LIN {X 0,Y 262.907,Z 862.683,A -85,B 0,C 180,E1 12997.239,E2 12997.239} C_VEL
LIN {X 0,Y 257.148,Z 985.55,A -85,B 0,C 180,E1 12992.155,E2 12992.155} C_VEL
LIN {X 0,Y 256.421,Z 1011.983,A -85,B 0,C 180,E1 12990.929,E2 12990.929} C_VEL
LIN {X 0,Y 255.607,Z 1029.219,A -85,B 0,C 180,E1 12989.732,E2 12989.732} C_VEL
LIN {X 0,Y 254.567,Z 1046.159,A -85,B 0,C 180,E1 12988.115,E2 12988.115} C_VEL
LIN {X 0,Y 253.439,Z 1061.43,A -85,B 0,C 180,E1 12986.217,E2 12986.217} C_VEL
LIN {X 0,Y 252.31,Z 1075.854,A -85,B 0,C 180,E1 12983.96,E2 12983.96} C_VEL
LIN {X 0,Y 251.242,Z 1089.802,A -85,B 0,C 180,E1 12981.227,E2 12981.227} C_VEL
LIN {X 0,Y 250.502,Z 1101.467,A -85,B 0,C 180,E1 12978.375,E2 12978.375} C_VEL
LIN {X 0,Y 250.09,Z 1111.696,A -85,B 0,C 180,E1 12975.295,E2 12975.295} C_VEL
LIN {X 0,Y 250.084,Z 1120.327,A -85,B 0,C 180,E1 12971.994,E2 12971.994} C_VEL
LIN {X 0,Y 250.563,Z 1126.995,A -85,B 0,C 180,E1 12968.717,E2 12968.717} C_VEL
LIN {X 0,Y 251.586,Z 1131.816,A -85,B 0,C 180,E1 12965.468,E2 12965.468} C_VEL
LIN {X 0,Y 253.23,Z 1135.281,A -85,B 0,C 180,E1 12962.258,E2 12962.258} C_VEL
LIN {X 0,Y 255.925,Z 1137.41,A -85,B 0,C 180,E1 12958.652,E2 12958.652} C_VEL
LIN {X 0,Y 259.509,Z 1137.615,A -85,B 0,C 180,E1 12955.133,E2 12955.133} C_VEL
LIN {X 0,Y 263.997,Z 1136.033,A -85,B 0,C 180,E1 12951.72,E2 12951.72} C_VEL
LIN {X 0,Y 265.449,Z 1135.191,A -85,B 0,C 180,E1 12950.758,E2 12950.758} C_VEL
LIN {X 0,Y 267.144,Z 1133.765,A -85,B 0,C 180,E1 12949.03,E2 12949.03} C_VEL
LIN {X 0,Y 268.599,Z 1130.246,A -85,B 0,C 180,E1 12945.292,E2 12945.292} C_VEL
LIN {X 0,Y 270.654,Z 1127.621,A -85,B 0,C 180,E1 12943.679,E2 12943.679} C_VEL
LIN {X 0,Y 271.079,Z 1127.193,A -85,B 0,C 180,E1 12943.483,E2 12943.483} C_VEL
LIN {X 0,Y 278.019,Z 1119.744,A -85,B 0,C 180,E1 12940.674,E2 12940.674} C_VEL
LIN {X 0,Y 285.046,Z 1110.662,A -85,B 0,C 180,E1 12938.167,E2 12938.167} C_VEL
LIN {X 0,Y 291.992,Z 1100.144,A -85,B 0,C 180,E1 12935.948,E2 12935.948} C_VEL
LIN {X 0,Y 298.978,Z 1087.604,A -85,B 0,C 180,E1 12933.906,E2 12933.906} C_VEL
LIN {X 0,Y 305.649,Z 1073.127,A -85,B 0,C 180,E1 12932.104,E2 12932.104} C_VEL
LIN {X 0,Y 310.7,Z 1059.737,A -85,B 0,C 180,E1 12930.816,E2 12930.816} C_VEL
LIN {X 0,Y 314.858,Z 1046.143,A -85,B 0,C 180,E1 12929.775,E2 12929.775} C_VEL
LIN {X 0,Y 318.495,Z 1031.06,A -85,B 0,C 180,E1 12928.863,E2 12928.863} C_VEL
LIN {X 0,Y 324.296,Z 999.248,A -85,B 0,C 180,E1 12927.506,E2 12927.506} C_VEL
LIN {X 0,Y 338.694,Z 926.288,A -85,B 0,C 180,E1 12925.071,E2 12925.071} C_VEL
LIN {X 0,Y 330.952,Z 955.979,A -85,B 0,C 180,E1 12923.859,E2 12923.859} C_VEL
LIN {X 0,Y 322.137,Z 991.386,A -85,B 0,C 180,E1 12922.542,E2 12922.542} C_VEL
LIN {X 0,Y 313.495,Z 1027.366,A -85,B 0,C 180,E1 12920.786,E2 12920.786} C_VEL
LIN {X 0,Y 308.225,Z 1048.269,A -85,B 0,C 180,E1 12919.544,E2 12919.544} C_VEL
LIN {X 0,Y 302.397,Z 1065.839,A -85,B 0,C 180,E1 12918.208,E2 12918.208} C_VEL
LIN {X 0,Y 295.952,Z 1082.262,A -85,B 0,C 180,E1 12916.721,E2 12916.721} C_VEL
LIN {X 0,Y 289.029,Z 1097.291,A -85,B 0,C 180,E1 12915.024,E2 12915.024} C_VEL
LIN {X 0,Y 281.432,Z 1112.235,A -85,B 0,C 180,E1 12912.868,E2 12912.868} C_VEL
LIN {X 0,Y 273.14,Z 1127.155,A -85,B 0,C 180,E1 12910.108,E2 12910.108} C_VEL
LIN {X 0,Y 265.471,Z 1140.112,A -85,B 0,C 180,E1 12907.054,E2 12907.054} C_VEL
LIN {X 0,Y 258.017,Z 1152.256,A -85,B 0,C 180,E1 12903.383,E2 12903.383} C_VEL
LIN {X 0,Y 251.919,Z 1162.119,A -85,B 0,C 180,E1 12899.479,E2 12899.479} C_VEL
LIN {X 0,Y 247.143,Z 1170.061,A -85,B 0,C 180,E1 12895.391,E2 12895.391} C_VEL
LIN {X 0,Y 243.863,Z 1176.091,A -85,B 0,C 180,E1 12891.147,E2 12891.147} C_VEL
LIN {X 0,Y 242.039,Z 1180.61,A -85,B 0,C 180,E1 12886.558,E2 12886.558} C_VEL
LIN {X 0,Y 241.078,Z 1189.876,A -85,B 0,C 180,E1 12881.965,E2 12881.965} C_VEL
LIN {X 0,Y 240.853,Z 1196.891,A -85,B 0,C 180,E1 12877.631,E2 12877.631} C_VEL
LIN {X 0,Y 240.925,Z 1201.889,A -85,B 0,C 180,E1 12873.566,E2 12873.566} C_VEL
LIN {X 0,Y 240.878,Z 1205.148,A -85,B 0,C 180,E1 12869.997,E2 12869.997} C_VEL
LIN {X 0,Y 240.501,Z 1207.636,A -85,B 0,C 180,E1 12865.944,E2 12865.944} C_VEL
LIN {X 0,Y 240.266,Z 1209.075,A -85,B 0,C 180,E1 12860.898,E2 12860.898} C_VEL
LIN {X 0,Y 241.096,Z 1209.016,A -85,B 0,C 180,E1 12855.588,E2 12855.588} C_VEL
LIN {X 0,Y 243.908,Z 1207.154,A -85,B 0,C 180,E1 12849.855,E2 12849.855} C_VEL
LIN {X 0,Y 249.522,Z 1203.368,A -85,B 0,C 180,E1 12843.842,E2 12843.842} C_VEL
LIN {X 0,Y 258.306,Z 1197.619,A -85,B 0,C 180,E1 12837.97,E2 12837.97} C_VEL
LIN {X 0,Y 270.003,Z 1190.061,A -85,B 0,C 180,E1 12832.6,E2 12832.6} C_VEL
LIN {X 0,Y 285.633,Z 1180.278,A -85,B 0,C 180,E1 12827.495,E2 12827.495} C_VEL
LIN {X 0,Y 303.551,Z 1169.347,A -85,B 0,C 180,E1 12823.252,E2 12823.252} C_VEL
LIN {X 0,Y 286.385,Z 1177.494,A -85,B 0,C 180,E1 12818.941,E2 12818.941} C_VEL
LIN {X 0,Y 272.266,Z 1183.771,A -85,B 0,C 180,E1 12814.191,E2 12814.191} C_VEL
LIN {X 0,Y 260.321,Z 1188.527,A -85,B 0,C 180,E1 12808.698,E2 12808.698} C_VEL
LIN {X 0,Y 251.821,Z 1191.239,A -85,B 0,C 180,E1 12803.152,E2 12803.152} C_VEL
LIN {X 0,Y 246.032,Z 1192.182,A -85,B 0,C 180,E1 12797.507,E2 12797.507} C_VEL
LIN {X 0,Y 242.552,Z 1191.319,A -85,B 0,C 180,E1 12791.9,E2 12791.9} C_VEL
LIN {X 0,Y 240.867,Z 1188.892,A -85,B 0,C 180,E1 12786.44,E2 12786.44} C_VEL
LIN {X 0,Y 240.315,Z 1185.407,A -85,B 0,C 180,E1 12781.674,E2 12781.674} C_VEL
LIN {X 0,Y 240.198,Z 1180.652,A -85,B 0,C 180,E1 12777.142,E2 12777.142} C_VEL
LIN {X 0,Y 240.391,Z 1174.513,A -85,B 0,C 180,E1 12772.597,E2 12772.597} C_VEL
LIN {X 0,Y 241.092,Z 1166.593,A -85,B 0,C 180,E1 12768.037,E2 12768.037} C_VEL
LIN {X 0,Y 242.519,Z 1156.908,A -85,B 0,C 180,E1 12763.478,E2 12763.478} C_VEL
LIN {X 0,Y 244.727,Z 1145.903,A -85,B 0,C 180,E1 12759.184,E2 12759.184} C_VEL
LIN {X 0,Y 247.867,Z 1132.744,A -85,B 0,C 180,E1 12754.946,E2 12754.946} C_VEL
LIN {X 0,Y 251.721,Z 1118.125,A -85,B 0,C 180,E1 12751.019,E2 12751.019} C_VEL
LIN {X 0,Y 256.476,Z 1101.03,A -85,B 0,C 180,E1 12747.193,E2 12747.193} C_VEL
LIN {X 0,Y 261.576,Z 1082.796,A -85,B 0,C 180,E1 12743.808,E2 12743.808} C_VEL
LIN {X 0,Y 266.72,Z 1063.992,A -85,B 0,C 180,E1 12740.9,E2 12740.9} C_VEL
LIN {X 0,Y 272.079,Z 1043.302,A -85,B 0,C 180,E1 12738.25,E2 12738.25} C_VEL
LIN {X 0,Y 277.383,Z 1021.009,A -85,B 0,C 180,E1 12735.923,E2 12735.923} C_VEL
LIN {X 0,Y 282.447,Z 997.128,A -85,B 0,C 180,E1 12733.919,E2 12733.919} C_VEL
LIN {X 0,Y 286.934,Z 972.487,A -85,B 0,C 180,E1 12732.294,E2 12732.294} C_VEL
LIN {X 0,Y 290.636,Z 947.66,A -85,B 0,C 180,E1 12731.044,E2 12731.044} C_VEL
LIN {X 0,Y 297.427,Z 889.487,A -85,B 0,C 180,E1 12728.954,E2 12728.954} C_VEL
LIN {X 0,Y 310.27,Z 781.665,A -85,B 0,C 180,E1 12725.402,E2 12725.402} C_VEL
LIN {X 0,Y 296.592,Z 756.31,A -85,B 0,C 180,E1 12722.045,E2 12722.045} C_VEL
LIN {X 0,Y 283.156,Z 732.602,A -85,B 0,C 180,E1 12718.388,E2 12718.388} C_VEL
LIN {X 0,Y 271.277,Z 712.791,A -85,B 0,C 180,E1 12714.82,E2 12714.82} C_VEL
LIN {X 0,Y 260.212,Z 695.463,A -85,B 0,C 180,E1 12711.177,E2 12711.177} C_VEL
LIN {X 0,Y 252.89,Z 684.704,A -85,B 0,C 180,E1 12708.562,E2 12708.562} C_VEL
LIN {X 0,Y 250.262,Z 680.677,A -85,B 0,C 180,E1 12707.56,E2 12707.56} C_VEL
LIN {X 0,Y 247.641,Z 676.731,A -85,B 0,C 180,E1 12706.541,E2 12706.541} C_VEL
LIN {X 0,Y 246.731,Z 675.484,A -85,B 0,C 180,E1 12706.19,E2 12706.19} C_VEL
LIN {X 0,Y 244.47,Z 672.459,A -85,B 0,C 180,E1 12705.299,E2 12705.299} C_VEL
LIN {X 0,Y 243.869,Z 670.279,A -85,B 0,C 180,E1 12704.912,E2 12704.912} C_VEL
LIN {X 0,Y 243.87,Z 670.278,A -85,B 0,C 180,E1 12699.919,E2 12699.919} C_VEL
LIN {X 0,Y 243.842,Z 670.293,A -85,B 0,C 180,E1 12694.943,E2 12694.943} C_VEL
LIN {X 0,Y 243.858,Z 670.294,A -85,B 0,C 180,E1 12689.533,E2 12689.533} C_VEL
LIN {X 0,Y 243.883,Z 670.266,A -85,B 0,C 180,E1 12684.592,E2 12684.592} C_VEL
LIN {X 0,Y 243.852,Z 670.26,A -85,B 0,C 180,E1 12679.732,E2 12679.732} C_VEL
LIN {X 0,Y 243.847,Z 670.293,A -85,B 0,C 180,E1 12674.473,E2 12674.473} C_VEL
LIN {X 0,Y 243.873,Z 670.284,A -85,B 0,C 180,E1 12669.357,E2 12669.357} C_VEL
LIN {X 0,Y 243.901,Z 670.438,A -85,B 0,C 180,E1 12664.735,E2 12664.735} C_VEL
LIN {X 0,Y 251.948,Z 691.844,A -85,B 0,C 180,E1 12660.525,E2 12660.525} C_VEL
LIN {X 0,Y 259.45,Z 713.889,A -85,B 0,C 180,E1 12656.561,E2 12656.561} C_VEL
LIN {X 0,Y 265.405,Z 734.117,A -85,B 0,C 180,E1 12653.205,E2 12653.205} C_VEL
LIN {X 0,Y 268.217,Z 745.033,A -85,B 0,C 180,E1 12651.501,E2 12651.501} C_VEL
LIN {X 0,Y 263.398,Z 787.814,A -85,B 0,C 180,E1 12646.466,E2 12646.466} C_VEL
LIN {X 0,Y 258.769,Z 832.439,A -85,B 0,C 180,E1 12641.187,E2 12641.187} C_VEL
LIN {X 0,Y 256.454,Z 854.436,A -85,B 0,C 180,E1 12638.589,E2 12638.589} C_VEL
LIN {X 0,Y 255.062,Z 863.549,A -85,B 0,C 180,E1 12637.603,E2 12637.603} C_VEL
LIN {X 0,Y 249.206,Z 985.599,A -85,B 0,C 180,E1 12632.372,E2 12632.372} C_VEL
LIN {X 0,Y 248.442,Z 1012.462,A -85,B 0,C 180,E1 12631.085,E2 12631.085} C_VEL
LIN {X 0,Y 247.567,Z 1030.453,A -85,B 0,C 180,E1 12629.781,E2 12629.781} C_VEL
LIN {X 0,Y 246.475,Z 1047.618,A -85,B 0,C 180,E1 12628.066,E2 12628.066} C_VEL
LIN {X 0,Y 245.276,Z 1063.53,A -85,B 0,C 180,E1 12625.985,E2 12625.985} C_VEL
LIN {X 0,Y 244.151,Z 1077.714,A -85,B 0,C 180,E1 12623.656,E2 12623.656} C_VEL
LIN {X 0,Y 243.108,Z 1091.585,A -85,B 0,C 180,E1 12620.823,E2 12620.823} C_VEL
LIN {X 0,Y 242.37,Z 1103.934,A -85,B 0,C 180,E1 12617.653,E2 12617.653} C_VEL
LIN {X 0,Y 242.052,Z 1113.48,A -85,B 0,C 180,E1 12614.589,E2 12614.589} C_VEL
LIN {X 0,Y 242.18,Z 1122.496,A -85,B 0,C 180,E1 12610.943,E2 12610.943} C_VEL
LIN {X 0,Y 242.922,Z 1129.293,A -85,B 0,C 180,E1 12607.295,E2 12607.295} C_VEL
LIN {X 0,Y 244.855,Z 1135.134,A -85,B 0,C 180,E1 12602.804,E2 12602.804} C_VEL
LIN {X 0,Y 247.469,Z 1138.004,A -85,B 0,C 180,E1 12599.069,E2 12599.069} C_VEL
LIN {X 0,Y 251.021,Z 1138.959,A -85,B 0,C 180,E1 12595.426,E2 12595.426} C_VEL
LIN {X 0,Y 255.522,Z 1138.14,A -85,B 0,C 180,E1 12591.897,E2 12591.897} C_VEL
LIN {X 0,Y 260.921,Z 1135.403,A -85,B 0,C 180,E1 12588.501,E2 12588.501} C_VEL
LIN {X 0,Y 267.191,Z 1130.78,A -85,B 0,C 180,E1 12585.253,E2 12585.253} C_VEL
LIN {X 0,Y 271.079,Z 1127.193,A -85,B 0,C 180,E1 12583.483,E2 12583.483} C_VEL
LIN {X 0,Y 273.484,Z 1124.348,A -85,B 0,C 180,E1 12582.046,E2 12582.046} C_VEL
LIN {X 0,Y 276.801,Z 1117.935,A -85,B 0,C 180,E1 12578.641,E2 12578.641} C_VEL
LIN {X 0,Y 279.108,Z 1114.254,A -85,B 0,C 180,E1 12577.323,E2 12577.323} C_VEL
LIN {X 0,Y 280.012,Z 1113.013,A -85,B 0,C 180,E1 12576.996,E2 12576.996} C_VEL
LIN {X 0,Y 287.643,Z 1102.313,A -85,B 0,C 180,E1 12574.683,E2 12574.683} C_VEL
LIN {X 0,Y 295.58,Z 1088.93,A -85,B 0,C 180,E1 12572.496,E2 12572.496} C_VEL
LIN {X 0,Y 302.679,Z 1074.368,A -85,B 0,C 180,E1 12570.698,E2 12570.698} C_VEL
LIN {X 0,Y 308.206,Z 1060.379,A -85,B 0,C 180,E1 12569.376,E2 12569.376} C_VEL
LIN {X 0,Y 312.574,Z 1046.756,A -85,B 0,C 180,E1 12568.354,E2 12568.354} C_VEL
LIN {X 0,Y 316.312,Z 1031.971,A -85,B 0,C 180,E1 12567.477,E2 12567.477} C_VEL
LIN {X 0,Y 322.674,Z 999.089,A -85,B 0,C 180,E1 12566.094,E2 12566.094} C_VEL
LIN {X 0,Y 329.477,Z 965.638,A -85,B 0,C 180,E1 12564.944,E2 12564.944} C_VEL
LIN {X 0,Y 320.95,Z 998.547,A -85,B 0,C 180,E1 12563.705,E2 12563.705} C_VEL
LIN {X 0,Y 310.763,Z 1038.509,A -85,B 0,C 180,E1 12561.704,E2 12561.704} C_VEL
LIN {X 0,Y 304.982,Z 1056.587,A -85,B 0,C 180,E1 12560.537,E2 12560.537} C_VEL
LIN {X 0,Y 297.577,Z 1075.428,A -85,B 0,C 180,E1 12558.963,E2 12558.963} C_VEL
LIN {X 0,Y 289.988,Z 1091.402,A -85,B 0,C 180,E1 12557.4,E2 12557.4} C_VEL
LIN {X 0,Y 281.3,Z 1107.424,A -85,B 0,C 180,E1 12555.304,E2 12555.304} C_VEL
LIN {X 0,Y 272.98,Z 1121.409,A -85,B 0,C 180,E1 12552.94,E2 12552.94} C_VEL
LIN {X 0,Y 264.299,Z 1134.834,A -85,B 0,C 180,E1 12550.022,E2 12550.022} C_VEL
LIN {X 0,Y 256.114,Z 1146.895,A -85,B 0,C 180,E1 12546.674,E2 12546.674} C_VEL
LIN {X 0,Y 248.363,Z 1157.914,A -85,B 0,C 180,E1 12542.643,E2 12542.643} C_VEL
LIN {X 0,Y 242.49,Z 1166.352,A -85,B 0,C 180,E1 12538.555,E2 12538.555} C_VEL
LIN {X 0,Y 237.831,Z 1173.199,A -85,B 0,C 180,E1 12534.063,E2 12534.063} C_VEL
LIN {X 0,Y 235.02,Z 1177.94,A -85,B 0,C 180,E1 12529.636,E2 12529.636} C_VEL
LIN {X 0,Y 233.992,Z 1180.433,A -85,B 0,C 180,E1 12526.25,E2 12526.25} C_VEL
LIN {X 0,Y 233.086,Z 1189.823,A -85,B 0,C 180,E1 12521.377,E2 12521.377} C_VEL
LIN {X 0,Y 232.929,Z 1196.73,A -85,B 0,C 180,E1 12516.9,E2 12516.9} C_VEL
LIN {X 0,Y 233.016,Z 1201.587,A -85,B 0,C 180,E1 12512.702,E2 12512.702} C_VEL
LIN {X 0,Y 232.885,Z 1204.73,A -85,B 0,C 180,E1 12509.013,E2 12509.013} C_VEL
LIN {X 0,Y 232.433,Z 1207.231,A -85,B 0,C 180,E1 12504.566,E2 12504.566} C_VEL
LIN {X 0,Y 232.386,Z 1208.487,A -85,B 0,C 180,E1 12499.335,E2 12499.335} C_VEL
LIN {X 0,Y 233.79,Z 1208.316,A -85,B 0,C 180,E1 12493.601,E2 12493.601} C_VEL
LIN {X 0,Y 237.606,Z 1206.216,A -85,B 0,C 180,E1 12487.481,E2 12487.481} C_VEL
LIN {X 0,Y 244.668,Z 1202.141,A -85,B 0,C 180,E1 12481.166,E2 12481.166} C_VEL
LIN {X 0,Y 254.823,Z 1196.35,A -85,B 0,C 180,E1 12475.319,E2 12475.319} C_VEL
LIN {X 0,Y 268.434,Z 1188.583,A -85,B 0,C 180,E1 12469.876,E2 12469.876} C_VEL
LIN {X 0,Y 285.564,Z 1178.951,A -85,B 0,C 180,E1 12464.982,E2 12464.982} C_VEL
LIN {X 0,Y 293.426,Z 1174.599,A -85,B 0,C 180,E1 12463.175,E2 12463.175} C_VEL
LIN {X 0,Y 276.489,Z 1181.641,A -85,B 0,C 180,E1 12458.733,E2 12458.733} C_VEL
LIN {X 0,Y 262.024,Z 1187.123,A -85,B 0,C 180,E1 12453.6,E2 12453.6} C_VEL
LIN {X 0,Y 250.761,Z 1190.751,A -85,B 0,C 180,E1 12448.073,E2 12448.073} C_VEL
LIN {X 0,Y 242.54,Z 1192.595,A -85,B 0,C 180,E1 12442.294,E2 12442.294} C_VEL
LIN {X 0,Y 237.092,Z 1192.604,A -85,B 0,C 180,E1 12436.418,E2 12436.418} C_VEL
LIN {X 0,Y 233.992,Z 1190.949,A -85,B 0,C 180,E1 12430.593,E2 12430.593} C_VEL
LIN {X 0,Y 232.645,Z 1187.943,A -85,B 0,C 180,E1 12425.184,E2 12425.184} C_VEL
LIN {X 0,Y 232.26,Z 1183.944,A -85,B 0,C 180,E1 12420.499,E2 12420.499} C_VEL
LIN {X 0,Y 232.221,Z 1178.664,A -85,B 0,C 180,E1 12415.808,E2 12415.808} C_VEL
LIN {X 0,Y 232.535,Z 1172.134,A -85,B 0,C 180,E1 12411.35,E2 12411.35} C_VEL
LIN {X 0,Y 233.498,Z 1163.129,A -85,B 0,C 180,E1 12406.383,E2 12406.383} C_VEL
LIN {X 0,Y 235.289,Z 1152.65,A -85,B 0,C 180,E1 12401.677,E2 12401.677} C_VEL
LIN {X 0,Y 237.924,Z 1140.682,A -85,B 0,C 180,E1 12397.261,E2 12397.261} C_VEL
LIN {X 0,Y 241.318,Z 1127.356,A -85,B 0,C 180,E1 12393.158,E2 12393.158} C_VEL
LIN {X 0,Y 245.76,Z 1111.304,A -85,B 0,C 180,E1 12389.031,E2 12389.031} C_VEL
LIN {X 0,Y 250.677,Z 1094.143,A -85,B 0,C 180,E1 12385.366,E2 12385.366} C_VEL
LIN {X 0,Y 255.878,Z 1075.916,A -85,B 0,C 180,E1 12382.129,E2 12382.129} C_VEL
LIN {X 0,Y 261.644,Z 1054.884,A -85,B 0,C 180,E1 12379.058,E2 12379.058} C_VEL
LIN {X 0,Y 267.378,Z 1032.375,A -85,B 0,C 180,E1 12376.381,E2 12376.381} C_VEL
LIN {X 0,Y 272.795,Z 1009.003,A -85,B 0,C 180,E1 12374.143,E2 12374.143} C_VEL
LIN {X 0,Y 277.725,Z 984.619,A -85,B 0,C 180,E1 12372.289,E2 12372.289} C_VEL
LIN {X 0,Y 281.98,Z 959.598,A -85,B 0,C 180,E1 12370.819,E2 12370.819} C_VEL
LIN {X 0,Y 285.461,Z 933.761,A -85,B 0,C 180,E1 12369.699,E2 12369.699} C_VEL
LIN {X 0,Y 303.575,Z 784.388,A -85,B 0,C 180,E1 12364.573,E2 12364.573} C_VEL
LIN {X 0,Y 288.726,Z 756.795,A -85,B 0,C 180,E1 12360.778,E2 12360.778} C_VEL
LIN {X 0,Y 274.471,Z 731.706,A -85,B 0,C 180,E1 12356.682,E2 12356.682} C_VEL
LIN {X 0,Y 262.767,Z 712.512,A -85,B 0,C 180,E1 12352.971,E2 12352.971} C_VEL
LIN {X 0,Y 252.332,Z 696.388,A -85,B 0,C 180,E1 12349.325,E2 12349.325} C_VEL
LIN {X 0,Y 245.659,Z 686.526,A -85,B 0,C 180,E1 12346.8,E2 12346.8} C_VEL
LIN {X 0,Y 242.421,Z 681.711,A -85,B 0,C 180,E1 12345.493,E2 12345.493} C_VEL
LIN {X 0,Y 239.862,Z 677.766,A -85,B 0,C 180,E1 12344.395,E2 12344.395} C_VEL
LIN {X 0,Y 239.036,Z 676.628,A -85,B 0,C 180,E1 12344.044,E2 12344.044} C_VEL
LIN {X 0,Y 236.628,Z 673.64,A -85,B 0,C 180,E1 12343.038,E2 12343.038} C_VEL
LIN {X 0,Y 235.942,Z 671.261,A -85,B 0,C 180,E1 12342.593,E2 12342.593} C_VEL
LIN {X 0,Y 235.928,Z 671.262,A -85,B 0,C 180,E1 12337.308,E2 12337.308} C_VEL
LIN {X 0,Y 235.879,Z 671.259,A -85,B 0,C 180,E1 12332.19,E2 12332.19} C_VEL
LIN {X 0,Y 235.934,Z 671.254,A -85,B 0,C 180,E1 12327.331,E2 12327.331} C_VEL
LIN {X 0,Y 235.949,Z 671.278,A -85,B 0,C 180,E1 12322.21,E2 12322.21} C_VEL
LIN {X 0,Y 235.905,Z 671.261,A -85,B 0,C 180,E1 12316.772,E2 12316.772} C_VEL
LIN {X 0,Y 235.916,Z 671.281,A -85,B 0,C 180,E1 12311.469,E2 12311.469} C_VEL
LIN {X 0,Y 235.952,Z 671.272,A -85,B 0,C 180,E1 12306.53,E2 12306.53} C_VEL
LIN {X 0,Y 235.972,Z 671.45,A -85,B 0,C 180,E1 12305.849,E2 12305.849} C_VEL
LIN {X 0,Y 243.869,Z 692.127,A -85,B 0,C 180,E1 12301.605,E2 12301.605} C_VEL
LIN {X 0,Y 251.152,Z 713.391,A -85,B 0,C 180,E1 12297.628,E2 12297.628} C_VEL
LIN {X 0,Y 257.574,Z 734.773,A -85,B 0,C 180,E1 12293.981,E2 12293.981} C_VEL
LIN {X 0,Y 260.697,Z 747.225,A -85,B 0,C 180,E1 12291.996,E2 12291.996} C_VEL
LIN {X 0,Y 255.647,Z 790.521,A -85,B 0,C 180,E1 12286.812,E2 12286.812} C_VEL
LIN {X 0,Y 250.873,Z 835.148,A -85,B 0,C 180,E1 12281.416,E2 12281.416} C_VEL
LIN {X 0,Y 248.798,Z 854.259,A -85,B 0,C 180,E1 12279.114,E2 12279.114} C_VEL
LIN {X 0,Y 247.229,Z 864.336,A -85,B 0,C 180,E1 12277.99,E2 12277.99} C_VEL
LIN {X 0,Y 241.255,Z 985.467,A -85,B 0,C 180,E1 12272.577,E2 12272.577} C_VEL
LIN {X 0,Y 240.415,Z 1013.694,A -85,B 0,C 180,E1 12271.16,E2 12271.16} C_VEL
LIN {X 0,Y 239.54,Z 1031.22,A -85,B 0,C 180,E1 12269.846,E2 12269.846} C_VEL
LIN {X 0,Y 238.384,Z 1048.948,A -85,B 0,C 180,E1 12268.013,E2 12268.013} C_VEL
LIN {X 0,Y 237.109,Z 1065.635,A -85,B 0,C 180,E1 12265.738,E2 12265.738} C_VEL
LIN {X 0,Y 235.94,Z 1080.241,A -85,B 0,C 180,E1 12263.205,E2 12263.205} C_VEL
LIN {X 0,Y 235.048,Z 1092.259,A -85,B 0,C 180,E1 12260.642,E2 12260.642} C_VEL
LIN {X 0,Y 234.333,Z 1104.572,A -85,B 0,C 180,E1 12257.373,E2 12257.373} C_VEL
LIN {X 0,Y 234.04,Z 1114.526,A -85,B 0,C 180,E1 12254.089,E2 12254.089} C_VEL
LIN {X 0,Y 234.256,Z 1123.525,A -85,B 0,C 180,E1 12250.322,E2 12250.322} C_VEL
LIN {X 0,Y 235.12,Z 1130.307,A -85,B 0,C 180,E1 12246.588,E2 12246.588} C_VEL
LIN {X 0,Y 237.163,Z 1135.991,A -85,B 0,C 180,E1 12242.169,E2 12242.169} C_VEL
LIN {X 0,Y 240.07,Z 1139.072,A -85,B 0,C 180,E1 12238.23,E2 12238.23} C_VEL
LIN {X 0,Y 243.806,Z 1140.18,A -85,B 0,C 180,E1 12234.582,E2 12234.582} C_VEL
LIN {X 0,Y 248.941,Z 1139.436,A -85,B 0,C 180,E1 12230.75,E2 12230.75} C_VEL
LIN {X 0,Y 254.74,Z 1136.817,A -85,B 0,C 180,E1 12227.298,E2 12227.298} C_VEL
LIN {X 0,Y 261.427,Z 1132.299,A -85,B 0,C 180,E1 12224.011,E2 12224.011} C_VEL
LIN {X 0,Y 268.53,Z 1126.01,A -85,B 0,C 180,E1 12221.035,E2 12221.035} C_VEL
LIN {X 0,Y 276.036,Z 1117.959,A -85,B 0,C 180,E1 12218.312,E2 12218.312} C_VEL
LIN {X 0,Y 280.012,Z 1113.013,A -85,B 0,C 180,E1 12216.996,E2 12216.996} C_VEL
LIN {X 0,Y 282.808,Z 1108.817,A -85,B 0,C 180,E1 12215.79,E2 12215.79} C_VEL
LIN {X 0,Y 287.578,Z 1099.088,A -85,B 0,C 180,E1 12212.659,E2 12212.659} C_VEL
LIN {X 0,Y 290.233,Z 1094.147,A -85,B 0,C 180,E1 12211.611,E2 12211.611} C_VEL
LIN {X 0,Y 290.692,Z 1093.356,A -85,B 0,C 180,E1 12211.488,E2 12211.488} C_VEL
LIN {X 0,Y 297.857,Z 1080.218,A -85,B 0,C 180,E1 12209.761,E2 12209.761} C_VEL
LIN {X 0,Y 304.423,Z 1065.555,A -85,B 0,C 180,E1 12208.281,E2 12208.281} C_VEL
LIN {X 0,Y 309.941,Z 1049.888,A -85,B 0,C 180,E1 12207.068,E2 12207.068} C_VEL
LIN {X 0,Y 314.188,Z 1034.393,A -85,B 0,C 180,E1 12206.139,E2 12206.139} C_VEL
LIN {X 0,Y 320.128,Z 1005.276,A -85,B 0,C 180,E1 12204.878,E2 12204.878} C_VEL
LIN {X 0,Y 310.483,Z 1040.523,A -85,B 0,C 180,E1 12203.132,E2 12203.132} C_VEL
LIN {X 0,Y 303.258,Z 1060.576,A -85,B 0,C 180,E1 12201.842,E2 12201.842} C_VEL
LIN {X 0,Y 295.782,Z 1077.535,A -85,B 0,C 180,E1 12200.416,E2 12200.416} C_VEL
LIN {X 0,Y 287.08,Z 1094.008,A -85,B 0,C 180,E1 12198.787,E2 12198.787} C_VEL
LIN {X 0,Y 278.266,Z 1108.769,A -85,B 0,C 180,E1 12196.834,E2 12196.834} C_VEL
LIN {X 0,Y 268.806,Z 1123.001,A -85,B 0,C 180,E1 12194.367,E2 12194.367} C_VEL
LIN {X 0,Y 259.595,Z 1135.874,A -85,B 0,C 180,E1 12191.486,E2 12191.486} C_VEL
LIN {X 0,Y 250.356,Z 1147.937,A -85,B 0,C 180,E1 12187.951,E2 12187.951} C_VEL
LIN {X 0,Y 242.443,Z 1157.88,A -85,B 0,C 180,E1 12184.113,E2 12184.113} C_VEL
LIN {X 0,Y 235.723,Z 1166.284,A -85,B 0,C 180,E1 12179.751,E2 12179.751} C_VEL
LIN {X 0,Y 230.795,Z 1172.484,A -85,B 0,C 180,E1 12175.394,E2 12175.394} C_VEL
LIN {X 0,Y 227.366,Z 1177.205,A -85,B 0,C 180,E1 12170.481,E2 12170.481} C_VEL
LIN {X 0,Y 225.99,Z 1179.925,A -85,B 0,C 180,E1 12166.049,E2 12166.049} C_VEL
LIN {X 0,Y 225.133,Z 1189.293,A -85,B 0,C 180,E1 12161.006,E2 12161.006} C_VEL
LIN {X 0,Y 225.025,Z 1196.176,A -85,B 0,C 180,E1 12156.374,E2 12156.374} C_VEL
LIN {X 0,Y 225.106,Z 1200.991,A -85,B 0,C 180,E1 12152.033,E2 12152.033} C_VEL
LIN {X 0,Y 224.924,Z 1203.915,A -85,B 0,C 180,E1 12148.468,E2 12148.468} C_VEL
LIN {X 0,Y 224.496,Z 1206.198,A -85,B 0,C 180,E1 12144.373,E2 12144.373} C_VEL
LIN {X 0,Y 224.487,Z 1207.793,A -85,B 0,C 180,E1 12138.695,E2 12138.695} C_VEL
LIN {X 0,Y 226.12,Z 1207.743,A -85,B 0,C 180,E1 12132.763,E2 12132.763} C_VEL
LIN {X 0,Y 230.547,Z 1205.851,A -85,B 0,C 180,E1 12126.209,E2 12126.209} C_VEL
LIN {X 0,Y 238.008,Z 1202.241,A -85,B 0,C 180,E1 12119.939,E2 12119.939} C_VEL
LIN {X 0,Y 249.157,Z 1196.592,A -85,B 0,C 180,E1 12113.845,E2 12113.845} C_VEL
LIN {X 0,Y 264.125,Z 1189.004,A -85,B 0,C 180,E1 12108.217,E2 12108.217} C_VEL
LIN {X 0,Y 282.13,Z 1179.932,A -85,B 0,C 180,E1 12103.4,E2 12103.4} C_VEL
LIN {X 0,Y 283.219,Z 1179.348,A -85,B 0,C 180,E1 12103.095,E2 12103.095} C_VEL
LIN {X 0,Y 265.988,Z 1185.521,A -85,B 0,C 180,E1 12098.34,E2 12098.34} C_VEL
LIN {X 0,Y 251.315,Z 1190.094,A -85,B 0,C 180,E1 12092.763,E2 12092.763} C_VEL
LIN {X 0,Y 240.489,Z 1192.678,A -85,B 0,C 180,E1 12086.954,E2 12086.954} C_VEL
LIN {X 0,Y 232.796,Z 1193.51,A -85,B 0,C 180,E1 12080.89,E2 12080.89} C_VEL
LIN {X 0,Y 227.918,Z 1192.519,A -85,B 0,C 180,E1 12074.746,E2 12074.746} C_VEL
LIN {X 0,Y 225.35,Z 1189.906,A -85,B 0,C 180,E1 12068.682,E2 12068.682} C_VEL
LIN {X 0,Y 224.434,Z 1186.205,A -85,B 0,C 180,E1 12063.326,E2 12063.326} C_VEL
LIN {X 0,Y 224.222,Z 1181.383,A -85,B 0,C 180,E1 12058.472,E2 12058.472} C_VEL
LIN {X 0,Y 224.325,Z 1175.406,A -85,B 0,C 180,E1 12053.734,E2 12053.734} C_VEL
LIN {X 0,Y 224.893,Z 1167.752,A -85,B 0,C 180,E1 12048.984,E2 12048.984} C_VEL
LIN {X 0,Y 226.231,Z 1158.168,A -85,B 0,C 180,E1 12044.102,E2 12044.102} C_VEL
LIN {X 0,Y 228.391,Z 1147.25,A -85,B 0,C 180,E1 12039.504,E2 12039.504} C_VEL
LIN {X 0,Y 231.55,Z 1134.19,A -85,B 0,C 180,E1 12034.971,E2 12034.971} C_VEL
LIN {X 0,Y 235.489,Z 1119.73,A -85,B 0,C 180,E1 12030.778,E2 12030.778} C_VEL
LIN {X 0,Y 240.071,Z 1103.905,A -85,B 0,C 180,E1 12026.94,E2 12026.94} C_VEL
LIN {X 0,Y 245.306,Z 1086.063,A -85,B 0,C 180,E1 12023.341,E2 12023.341} C_VEL
LIN {X 0,Y 250.914,Z 1066.589,A -85,B 0,C 180,E1 12020.098,E2 12020.098} C_VEL
LIN {X 0,Y 256.66,Z 1045.514,A -85,B 0,C 180,E1 12017.218,E2 12017.218} C_VEL
LIN {X 0,Y 262.11,Z 1023.924,A -85,B 0,C 180,E1 12014.81,E2 12014.81} C_VEL
LIN {X 0,Y 267.116,Z 1001.827,A -85,B 0,C 180,E1 12012.812,E2 12012.812} C_VEL
LIN {X 0,Y 271.885,Z 977.755,A -85,B 0,C 180,E1 12011.078,E2 12011.078} C_VEL
LIN {X 0,Y 275.985,Z 952.789,A -85,B 0,C 180,E1 12009.691,E2 12009.691} C_VEL
LIN {X 0,Y 280.306,Z 919.414,A -85,B 0,C 180,E1 12008.343,E2 12008.343} C_VEL
LIN {X 0,Y 296.908,Z 787.157,A -85,B 0,C 180,E1 12003.73,E2 12003.73} C_VEL
LIN {X 0,Y 282.379,Z 760.081,A -85,B 0,C 180,E1 11999.867,E2 11999.867} C_VEL
LIN {X 0,Y 269.087,Z 736.594,A -85,B 0,C 180,E1 11995.944,E2 11995.944} C_VEL
LIN {X 0,Y 257.194,Z 716.769,A -85,B 0,C 180,E1 11992.007,E2 11992.007} C_VEL
LIN {X 0,Y 246.834,Z 700.863,A -85,B 0,C 180,E1 11988.269,E2 11988.269} C_VEL
LIN {X 0,Y 241.101,Z 692.304,A -85,B 0,C 180,E1 11986.012,E2 11986.012} C_VEL
LIN {X 0,Y 237.894,Z 687.556,A -85,B 0,C 180,E1 11984.672,E2 11984.672} C_VEL
LIN {X 0,Y 234.883,Z 683.027,A -85,B 0,C 180,E1 11983.356,E2 11983.356} C_VEL
LIN {X 0,Y 232.17,Z 679.267,A -85,B 0,C 180,E1 11982.175,E2 11982.175} C_VEL
LIN {X 0,Y 231.515,Z 677.932,A -85,B 0,C 180,E1 11981.841,E2 11981.841} C_VEL
LIN {X 0,Y 228.958,Z 675.18,A -85,B 0,C 180,E1 11980.738,E2 11980.738} C_VEL
LIN {X 0,Y 227.994,Z 672.257,A -85,B 0,C 180,E1 11980.107,E2 11980.107} C_VEL
LIN {X 0,Y 227.966,Z 672.271,A -85,B 0,C 180,E1 11975.036,E2 11975.036} C_VEL
LIN {X 0,Y 227.981,Z 672.272,A -85,B 0,C 180,E1 11969.501,E2 11969.501} C_VEL
LIN {X 0,Y 228.006,Z 672.247,A -85,B 0,C 180,E1 11964.215,E2 11964.215} C_VEL
LIN {X 0,Y 227.972,Z 672.232,A -85,B 0,C 180,E1 11959.133,E2 11959.133} C_VEL
LIN {X 0,Y 227.952,Z 672.269,A -85,B 0,C 180,E1 11953.844,E2 11953.844} C_VEL
LIN {X 0,Y 228.015,Z 672.263,A -85,B 0,C 180,E1 11948.66,E2 11948.66} C_VEL
LIN {X 0,Y 228.049,Z 672.5,A -85,B 0,C 180,E1 11946.968,E2 11946.968} C_VEL
LIN {X 0,Y 235.524,Z 691.848,A -85,B 0,C 180,E1 11942.851,E2 11942.851} C_VEL
LIN {X 0,Y 242.717,Z 712.355,A -85,B 0,C 180,E1 11938.873,E2 11938.873} C_VEL
LIN {X 0,Y 249.299,Z 733.98,A -85,B 0,C 180,E1 11935.007,E2 11935.007} C_VEL
LIN {X 0,Y 253.186,Z 749.118,A -85,B 0,C 180,E1 11932.532,E2 11932.532} C_VEL
LIN {X 0,Y 248.012,Z 792.076,A -85,B 0,C 180,E1 11927.303,E2 11927.303} C_VEL
LIN {X 0,Y 243.193,Z 835.777,A -85,B 0,C 180,E1 11921.917,E2 11921.917} C_VEL
LIN {X 0,Y 240.984,Z 855.002,A -85,B 0,C 180,E1 11919.553,E2 11919.553} C_VEL
LIN {X 0,Y 239.373,Z 865.29,A -85,B 0,C 180,E1 11918.369,E2 11918.369} C_VEL
LIN {X 0,Y 233.3,Z 985.346,A -85,B 0,C 180,E1 11912.78,E2 11912.78} C_VEL
LIN {X 0,Y 232.403,Z 1014.546,A -85,B 0,C 180,E1 11911.266,E2 11911.266} C_VEL
LIN {X 0,Y 231.513,Z 1031.984,A -85,B 0,C 180,E1 11909.916,E2 11909.916} C_VEL
LIN {X 0,Y 230.364,Z 1049.278,A -85,B 0,C 180,E1 11908.077,E2 11908.077} C_VEL
LIN {X 0,Y 229.228,Z 1064.015,A -85,B 0,C 180,E1 11906.039,E2 11906.039} C_VEL
LIN {X 0,Y 228.049,Z 1078.654,A -85,B 0,C 180,E1 11903.509,E2 11903.509} C_VEL
LIN {X 0,Y 226.972,Z 1093.139,A -85,B 0,C 180,E1 11900.36,E2 11900.36} C_VEL
LIN {X 0,Y 226.319,Z 1104.698,A -85,B 0,C 180,E1 11897.212,E2 11897.212} C_VEL
LIN {X 0,Y 226.045,Z 1114.824,A -85,B 0,C 180,E1 11893.814,E2 11893.814} C_VEL
LIN {X 0,Y 226.314,Z 1123.969,A -85,B 0,C 180,E1 11889.916,E2 11889.916} C_VEL
LIN {X 0,Y 227.273,Z 1130.932,A -85,B 0,C 180,E1 11886.055,E2 11886.055} C_VEL
LIN {X 0,Y 229.344,Z 1136.576,A -85,B 0,C 180,E1 11881.743,E2 11881.743} C_VEL
LIN {X 0,Y 232.328,Z 1139.86,A -85,B 0,C 180,E1 11877.775,E2 11877.775} C_VEL
LIN {X 0,Y 236.362,Z 1141.36,A -85,B 0,C 180,E1 11873.924,E2 11873.924} C_VEL
LIN {X 0,Y 241.511,Z 1140.993,A -85,B 0,C 180,E1 11870.158,E2 11870.158} C_VEL
LIN {X 0,Y 247.872,Z 1138.698,A -85,B 0,C 180,E1 11866.464,E2 11866.464} C_VEL
LIN {X 0,Y 254.872,Z 1134.512,A -85,B 0,C 180,E1 11863.119,E2 11863.119} C_VEL
LIN {X 0,Y 262.19,Z 1128.787,A -85,B 0,C 180,E1 11860.154,E2 11860.154} C_VEL
LIN {X 0,Y 269.598,Z 1121.617,A -85,B 0,C 180,E1 11857.537,E2 11857.537} C_VEL
LIN {X 0,Y 277.534,Z 1112.512,A -85,B 0,C 180,E1 11855.065,E2 11855.065} C_VEL
LIN {X 0,Y 285.337,Z 1101.825,A -85,B 0,C 180,E1 11852.875,E2 11852.875} C_VEL
LIN {X 0,Y 290.692,Z 1093.356,A -85,B 0,C 180,E1 11851.488,E2 11851.488} C_VEL
LIN {X 0,Y 293.544,Z 1088.034,A -85,B 0,C 180,E1 11850.525,E2 11850.525} C_VEL
LIN {X 0,Y 298.671,Z 1075.769,A -85,B 0,C 180,E1 11847.907,E2 11847.907} C_VEL
LIN {X 0,Y 301.121,Z 1069.846,A -85,B 0,C 180,E1 11847.092,E2 11847.092} C_VEL
LIN {X 0,Y 301.51,Z 1068.926,A -85,B 0,C 180,E1 11847.004,E2 11847.004} C_VEL
LIN {X 0,Y 307.88,Z 1052.227,A -85,B 0,C 180,E1 11845.7,E2 11845.7} C_VEL
LIN {X 0,Y 312.127,Z 1037.834,A -85,B 0,C 180,E1 11844.808,E2 11844.808} C_VEL
LIN {X 0,Y 304.357,Z 1058.477,A -85,B 0,C 180,E1 11843.594,E2 11843.594} C_VEL
LIN {X 0,Y 296.425,Z 1075.477,A -85,B 0,C 180,E1 11842.274,E2 11842.274} C_VEL
LIN {X 0,Y 285.819,Z 1094.335,A -85,B 0,C 180,E1 11840.473,E2 11840.473} C_VEL
LIN {X 0,Y 275.446,Z 1110.147,A -85,B 0,C 180,E1 11838.394,E2 11838.394} C_VEL
LIN {X 0,Y 265.469,Z 1123.854,A -85,B 0,C 180,E1 11836,E2 11836} C_VEL
LIN {X 0,Y 255.068,Z 1136.893,A -85,B 0,C 180,E1 11833.002,E2 11833.002} C_VEL
LIN {X 0,Y 245.755,Z 1147.835,A -85,B 0,C 180,E1 11829.696,E2 11829.696} C_VEL
LIN {X 0,Y 236.712,Z 1157.849,A -85,B 0,C 180,E1 11825.652,E2 11825.652} C_VEL
LIN {X 0,Y 229.526,Z 1165.716,A -85,B 0,C 180,E1 11821.36,E2 11821.36} C_VEL
LIN {X 0,Y 223.663,Z 1171.993,A -85,B 0,C 180,E1 11816.55,E2 11816.55} C_VEL
LIN {X 0,Y 219.902,Z 1176.325,A -85,B 0,C 180,E1 11811.607,E2 11811.607} C_VEL
LIN {X 0,Y 218.094,Z 1178.796,A -85,B 0,C 180,E1 11806.51,E2 11806.51} C_VEL
LIN {X 0,Y 218.032,Z 1179.087,A -85,B 0,C 180,E1 11805.967,E2 11805.967} C_VEL
LIN {X 0,Y 217.208,Z 1188.297,A -85,B 0,C 180,E1 11800.875,E2 11800.875} C_VEL
LIN {X 0,Y 217.126,Z 1194.866,A -85,B 0,C 180,E1 11796.342,E2 11796.342} C_VEL
LIN {X 0,Y 217.204,Z 1199.885,A -85,B 0,C 180,E1 11791.843,E2 11791.843} C_VEL
LIN {X 0,Y 216.96,Z 1203.067,A -85,B 0,C 180,E1 11787.884,E2 11787.884} C_VEL
LIN {X 0,Y 216.495,Z 1205.487,A -85,B 0,C 180,E1 11783.366,E2 11783.366} C_VEL
LIN {X 0,Y 216.699,Z 1207.126,A -85,B 0,C 180,E1 11777.471,E2 11777.471} C_VEL
LIN {X 0,Y 218.903,Z 1207.081,A -85,B 0,C 180,E1 11771.073,E2 11771.073} C_VEL
LIN {X 0,Y 224.38,Z 1205.178,A -85,B 0,C 180,E1 11764.102,E2 11764.102} C_VEL
LIN {X 0,Y 233.176,Z 1201.537,A -85,B 0,C 180,E1 11757.584,E2 11757.584} C_VEL
LIN {X 0,Y 245.657,Z 1195.97,A -85,B 0,C 180,E1 11751.479,E2 11751.479} C_VEL
LIN {X 0,Y 261.885,Z 1188.652,A -85,B 0,C 180,E1 11745.979,E2 11745.979} C_VEL
LIN {X 0,Y 273.122,Z 1183.535,A -85,B 0,C 180,E1 11743.054,E2 11743.054} C_VEL
LIN {X 0,Y 256.015,Z 1188.715,A -85,B 0,C 180,E1 11738.109,E2 11738.109} C_VEL
LIN {X 0,Y 241.964,Z 1192.229,A -85,B 0,C 180,E1 11732.499,E2 11732.499} C_VEL
LIN {X 0,Y 231.286,Z 1193.999,A -85,B 0,C 180,E1 11726.447,E2 11726.447} C_VEL
LIN {X 0,Y 223.832,Z 1193.932,A -85,B 0,C 180,E1 11720.124,E2 11720.124} C_VEL
LIN {X 0,Y 219.268,Z 1192.198,A -85,B 0,C 180,E1 11713.723,E2 11713.723} C_VEL
LIN {X 0,Y 217.094,Z 1189.066,A -85,B 0,C 180,E1 11707.681,E2 11707.681} C_VEL
LIN {X 0,Y 216.374,Z 1184.875,A -85,B 0,C 180,E1 11702.389,E2 11702.389} C_VEL
LIN {X 0,Y 216.228,Z 1179.541,A -85,B 0,C 180,E1 11697.288,E2 11697.288} C_VEL
LIN {X 0,Y 216.43,Z 1173.153,A -85,B 0,C 180,E1 11692.573,E2 11692.573} C_VEL
LIN {X 0,Y 217.211,Z 1164.734,A -85,B 0,C 180,E1 11687.511,E2 11687.511} C_VEL
LIN {X 0,Y 218.745,Z 1155.003,A -85,B 0,C 180,E1 11682.722,E2 11682.722} C_VEL
LIN {X 0,Y 221.328,Z 1142.99,A -85,B 0,C 180,E1 11677.846,E2 11677.846} C_VEL
LIN {X 0,Y 225.031,Z 1128.743,A -85,B 0,C 180,E1 11673.056,E2 11673.056} C_VEL
LIN {X 0,Y 229.448,Z 1113.319,A -85,B 0,C 180,E1 11668.77,E2 11668.77} C_VEL
LIN {X 0,Y 234.509,Z 1096.404,A -85,B 0,C 180,E1 11664.865,E2 11664.865} C_VEL
LIN {X 0,Y 240.275,Z 1077.145,A -85,B 0,C 180,E1 11661.203,E2 11661.203} C_VEL
LIN {X 0,Y 246.198,Z 1056.59,A -85,B 0,C 180,E1 11658.01,E2 11658.01} C_VEL
LIN {X 0,Y 251.828,Z 1035.677,A -85,B 0,C 180,E1 11655.357,E2 11655.357} C_VEL
LIN {X 0,Y 257.294,Z 1013.57,A -85,B 0,C 180,E1 11653.072,E2 11653.072} C_VEL
LIN {X 0,Y 262.439,Z 990.065,A -85,B 0,C 180,E1 11651.121,E2 11651.121} C_VEL
LIN {X 0,Y 266.996,Z 965.55,A -85,B 0,C 180,E1 11649.524,E2 11649.524} C_VEL
LIN {X 0,Y 270.842,Z 940.368,A -85,B 0,C 180,E1 11648.293,E2 11648.293} C_VEL
LIN {X 0,Y 290.228,Z 789.881,A -85,B 0,C 180,E1 11642.844,E2 11642.844} C_VEL
LIN {X 0,Y 276.69,Z 764.593,A -85,B 0,C 180,E1 11639.143,E2 11639.143} C_VEL
LIN {X 0,Y 264.017,Z 741.893,A -85,B 0,C 180,E1 11635.251,E2 11635.251} C_VEL
LIN {X 0,Y 252.39,Z 722.411,A -85,B 0,C 180,E1 11631.317,E2 11631.317} C_VEL
LIN {X 0,Y 240.879,Z 704.336,A -85,B 0,C 180,E1 11626.957,E2 11626.957} C_VEL
LIN {X 0,Y 233.358,Z 693.293,A -85,B 0,C 180,E1 11623.823,E2 11623.823} C_VEL
LIN {X 0,Y 230.452,Z 689.054,A -85,B 0,C 180,E1 11622.547,E2 11622.547} C_VEL
LIN {X 0,Y 227.121,Z 684.174,A -85,B 0,C 180,E1 11620.999,E2 11620.999} C_VEL
LIN {X 0,Y 224.476,Z 680.502,A -85,B 0,C 180,E1 11619.716,E2 11619.716} C_VEL
LIN {X 0,Y 223.661,Z 678.969,A -85,B 0,C 180,E1 11619.265,E2 11619.265} C_VEL
LIN {X 0,Y 220.989,Z 676.139,A -85,B 0,C 180,E1 11618.001,E2 11618.001} C_VEL
LIN {X 0,Y 220.051,Z 673.239,A -85,B 0,C 180,E1 11617.313,E2 11617.313} C_VEL
LIN {X 0,Y 220.006,Z 673.237,A -85,B 0,C 180,E1 11611.827,E2 11611.827} C_VEL
LIN {X 0,Y 220.056,Z 673.226,A -85,B 0,C 180,E1 11606.878,E2 11606.878} C_VEL
LIN {X 0,Y 220.055,Z 673.251,A -85,B 0,C 180,E1 11601.643,E2 11601.643} C_VEL
LIN {X 0,Y 220.018,Z 673.245,A -85,B 0,C 180,E1 11596.335,E2 11596.335} C_VEL
LIN {X 0,Y 220.058,Z 673.255,A -85,B 0,C 180,E1 11590.632,E2 11590.632} C_VEL
LIN {X 0,Y 220.1,Z 673.48,A -85,B 0,C 180,E1 11588.224,E2 11588.224} C_VEL
LIN {X 0,Y 228.029,Z 693.712,A -85,B 0,C 180,E1 11583.717,E2 11583.717} C_VEL
LIN {X 0,Y 234.909,Z 713.377,A -85,B 0,C 180,E1 11579.764,E2 11579.764} C_VEL
LIN {X 0,Y 241.071,Z 733.261,A -85,B 0,C 180,E1 11576.096,E2 11576.096} C_VEL
LIN {X 0,Y 245.678,Z 750.861,A -85,B 0,C 180,E1 11573.098,E2 11573.098} C_VEL
LIN {X 0,Y 240.323,Z 793.73,A -85,B 0,C 180,E1 11567.772,E2 11567.772} C_VEL
LIN {X 0,Y 235.278,Z 838.221,A -85,B 0,C 180,E1 11562.173,E2 11562.173} C_VEL
LIN {X 0,Y 233.193,Z 855.414,A -85,B 0,C 180,E1 11560.021,E2 11560.021} C_VEL
LIN {X 0,Y 231.517,Z 866.203,A -85,B 0,C 180,E1 11558.765,E2 11558.765} C_VEL
LIN {X 0,Y 225.344,Z 985.342,A -85,B 0,C 180,E1 11552.989,E2 11552.989} C_VEL
LIN {X 0,Y 224.399,Z 1015.128,A -85,B 0,C 180,E1 11551.387,E2 11551.387} C_VEL
LIN {X 0,Y 223.451,Z 1033.207,A -85,B 0,C 180,E1 11549.922,E2 11549.922} C_VEL
LIN {X 0,Y 222.265,Z 1050.55,A -85,B 0,C 180,E1 11547.99,E2 11547.99} C_VEL
LIN {X 0,Y 220.99,Z 1066.797,A -85,B 0,C 180,E1 11545.617,E2 11545.617} C_VEL
LIN {X 0,Y 219.849,Z 1080.932,A -85,B 0,C 180,E1 11543.018,E2 11543.018} C_VEL
LIN {X 0,Y 218.86,Z 1094.579,A -85,B 0,C 180,E1 11539.892,E2 11539.892} C_VEL
LIN {X 0,Y 218.212,Z 1107.334,A -85,B 0,C 180,E1 11536.225,E2 11536.225} C_VEL
LIN {X 0,Y 218.069,Z 1117.071,A -85,B 0,C 180,E1 11532.708,E2 11532.708} C_VEL
LIN {X 0,Y 218.53,Z 1125.979,A -85,B 0,C 180,E1 11528.679,E2 11528.679} C_VEL
LIN {X 0,Y 219.759,Z 1132.68,A -85,B 0,C 180,E1 11524.692,E2 11524.692} C_VEL
LIN {X 0,Y 222.588,Z 1138.609,A -85,B 0,C 180,E1 11519.737,E2 11519.737} C_VEL
LIN {X 0,Y 226.158,Z 1141.574,A -85,B 0,C 180,E1 11515.684,E2 11515.684} C_VEL
LIN {X 0,Y 230.815,Z 1142.669,A -85,B 0,C 180,E1 11511.776,E2 11511.776} C_VEL
LIN {X 0,Y 236.928,Z 1141.929,A -85,B 0,C 180,E1 11507.813,E2 11507.813} C_VEL
LIN {X 0,Y 243.691,Z 1139.311,A -85,B 0,C 180,E1 11504.283,E2 11504.283} C_VEL
LIN {X 0,Y 251.367,Z 1134.837,A -85,B 0,C 180,E1 11500.958,E2 11500.958} C_VEL
LIN {X 0,Y 259.278,Z 1128.729,A -85,B 0,C 180,E1 11498.028,E2 11498.028} C_VEL
LIN {X 0,Y 267.262,Z 1121.246,A -85,B 0,C 180,E1 11495.459,E2 11495.459} C_VEL
LIN {X 0,Y 275.112,Z 1112.483,A -85,B 0,C 180,E1 11493.209,E2 11493.209} C_VEL
LIN {X 0,Y 283.326,Z 1101.663,A -85,B 0,C 180,E1 11491.082,E2 11491.082} C_VEL
LIN {X 0,Y 291.533,Z 1088.712,A -85,B 0,C 180,E1 11489.149,E2 11489.149} C_VEL
LIN {X 0,Y 298.626,Z 1075.243,A -85,B 0,C 180,E1 11487.603,E2 11487.603} C_VEL
LIN {X 0,Y 301.51,Z 1068.926,A -85,B 0,C 180,E1 11487.004,E2 11487.004} C_VEL
LIN {X 0,Y 301.787,Z 1067.91,A -85,B 0,C 180,E1 11486.681,E2 11486.681} C_VEL
LIN {X 0,Y 301.159,Z 1068.309,A -85,B 0,C 180,E1 11486.029,E2 11486.029} C_VEL
LIN {X 0,Y 299.349,Z 1070.924,A -85,B 0,C 180,E1 11485.178,E2 11485.178} C_VEL
LIN {X 0,Y 295.978,Z 1076.64,A -85,B 0,C 180,E1 11484.219,E2 11484.219} C_VEL
LIN {X 0,Y 290.279,Z 1086.304,A -85,B 0,C 180,E1 11483.005,E2 11483.005} C_VEL
LIN {X 0,Y 287.339,Z 1091.006,A -85,B 0,C 180,E1 11482.533,E2 11482.533} C_VEL
LIN {X 0,Y 277.683,Z 1105.229,A -85,B 0,C 180,E1 11480.888,E2 11480.888} C_VEL
LIN {X 0,Y 267.179,Z 1118.92,A -85,B 0,C 180,E1 11478.778,E2 11478.778} C_VEL
LIN {X 0,Y 256.426,Z 1131.687,A -85,B 0,C 180,E1 11476.163,E2 11476.163} C_VEL
LIN {X 0,Y 245.953,Z 1143.044,A -85,B 0,C 180,E1 11473.072,E2 11473.072} C_VEL
LIN {X 0,Y 235.57,Z 1153.624,A -85,B 0,C 180,E1 11469.225,E2 11469.225} C_VEL
LIN {X 0,Y 226.756,Z 1162.09,A -85,B 0,C 180,E1 11464.972,E2 11464.972} C_VEL
LIN {X 0,Y 219.369,Z 1169.042,A -85,B 0,C 180,E1 11460.087,E2 11460.087} C_VEL
LIN {X 0,Y 214.206,Z 1173.788,A -85,B 0,C 180,E1 11455.132,E2 11455.132} C_VEL
LIN {X 0,Y 210.948,Z 1176.909,A -85,B 0,C 180,E1 11449.662,E2 11449.662} C_VEL
LIN {X 0,Y 210.106,Z 1177.997,A -85,B 0,C 180,E1 11445.972,E2 11445.972} C_VEL
LIN {X 0,Y 209.306,Z 1186.841,A -85,B 0,C 180,E1 11441.012,E2 11441.012} C_VEL
LIN {X 0,Y 209.237,Z 1193.581,A -85,B 0,C 180,E1 11436.248,E2 11436.248} C_VEL
LIN {X 0,Y 209.316,Z 1198.442,A -85,B 0,C 180,E1 11431.912,E2 11431.912} C_VEL
LIN {X 0,Y 209.052,Z 1201.852,A -85,B 0,C 180,E1 11427.803,E2 11427.803} C_VEL
LIN {X 0,Y 208.539,Z 1204.632,A -85,B 0,C 180,E1 11422.558,E2 11422.558} C_VEL
LIN {X 0,Y 208.878,Z 1206.294,A -85,B 0,C 180,E1 11416.713,E2 11416.713} C_VEL
LIN {X 0,Y 211.542,Z 1206.471,A -85,B 0,C 180,E1 11409.812,E2 11409.812} C_VEL
LIN {X 0,Y 217.364,Z 1204.96,A -85,B 0,C 180,E1 11402.905,E2 11402.905} C_VEL
LIN {X 0,Y 226.778,Z 1201.577,A -85,B 0,C 180,E1 11396.248,E2 11396.248} C_VEL
LIN {X 0,Y 241.02,Z 1196.074,A -85,B 0,C 180,E1 11389.667,E2 11389.667} C_VEL
LIN {X 0,Y 258.178,Z 1189.263,A -85,B 0,C 180,E1 11384.232,E2 11384.232} C_VEL
LIN {X 0,Y 262.887,Z 1187.266,A -85,B 0,C 180,E1 11382.995,E2 11382.995} C_VEL
LIN {X 0,Y 245.464,Z 1191.578,A -85,B 0,C 180,E1 11377.669,E2 11377.669} C_VEL
LIN {X 0,Y 231.681,Z 1194.119,A -85,B 0,C 180,E1 11371.76,E2 11371.76} C_VEL
LIN {X 0,Y 221.102,Z 1194.906,A -85,B 0,C 180,E1 11365.162,E2 11365.162} C_VEL
LIN {X 0,Y 214.254,Z 1193.837,A -85,B 0,C 180,E1 11358.508,E2 11358.508} C_VEL
LIN {X 0,Y 210.34,Z 1191.13,A -85,B 0,C 180,E1 11351.801,E2 11351.801} C_VEL
LIN {X 0,Y 208.733,Z 1187.285,A -85,B 0,C 180,E1 11345.779,E2 11345.779} C_VEL
LIN {X 0,Y 208.295,Z 1182.248,A -85,B 0,C 180,E1 11340.281,E2 11340.281} C_VEL
LIN {X 0,Y 208.284,Z 1176.488,A -85,B 0,C 180,E1 11335.325,E2 11335.325} C_VEL
LIN {X 0,Y 208.698,Z 1169.159,A -85,B 0,C 180,E1 11330.353,E2 11330.353} C_VEL
LIN {X 0,Y 209.863,Z 1159.774,A -85,B 0,C 180,E1 11325.098,E2 11325.098} C_VEL
LIN {X 0,Y 211.914,Z 1148.966,A -85,B 0,C 180,E1 11320.147,E2 11320.147} C_VEL
LIN {X 0,Y 215.028,Z 1136.146,A -85,B 0,C 180,E1 11315.267,E2 11315.267} C_VEL
LIN {X 0,Y 219.267,Z 1121.005,A -85,B 0,C 180,E1 11310.502,E2 11310.502} C_VEL
LIN {X 0,Y 224.163,Z 1104.76,A -85,B 0,C 180,E1 11306.273,E2 11306.273} C_VEL
LIN {X 0,Y 229.631,Z 1087.012,A -85,B 0,C 180,E1 11302.447,E2 11302.447} C_VEL
LIN {X 0,Y 235.71,Z 1066.874,A -85,B 0,C 180,E1 11298.897,E2 11298.897} C_VEL
LIN {X 0,Y 241.808,Z 1045.574,A -85,B 0,C 180,E1 11295.841,E2 11295.841} C_VEL
LIN {X 0,Y 247.722,Z 1023.224,A -85,B 0,C 180,E1 11293.243,E2 11293.243} C_VEL
LIN {X 0,Y 253.255,Z 999.857,A -85,B 0,C 180,E1 11291.062,E2 11291.062} C_VEL
LIN {X 0,Y 258.133,Z 976.11,A -85,B 0,C 180,E1 11289.318,E2 11289.318} C_VEL
LIN {X 0,Y 262.29,Z 951.705,A -85,B 0,C 180,E1 11287.933,E2 11287.933} C_VEL
LIN {X 0,Y 267.216,Z 915.317,A -85,B 0,C 180,E1 11286.425,E2 11286.425} C_VEL
LIN {X 0,Y 283.603,Z 792.774,A -85,B 0,C 180,E1 11281.96,E2 11281.96} C_VEL
LIN {X 0,Y 270.924,Z 768.847,A -85,B 0,C 180,E1 11278.343,E2 11278.343} C_VEL
LIN {X 0,Y 258.758,Z 746.953,A -85,B 0,C 180,E1 11274.517,E2 11274.517} C_VEL
LIN {X 0,Y 247.63,Z 728.053,A -85,B 0,C 180,E1 11270.6,E2 11270.6} C_VEL
LIN {X 0,Y 236.392,Z 710.237,A -85,B 0,C 180,E1 11266.214,E2 11266.214} C_VEL
LIN {X 0,Y 226.836,Z 695.899,A -85,B 0,C 180,E1 11262.039,E2 11262.039} C_VEL
LIN {X 0,Y 222.737,Z 690.158,A -85,B 0,C 180,E1 11260.086,E2 11260.086} C_VEL
LIN {X 0,Y 219.518,Z 685.42,A -85,B 0,C 180,E1 11258.451,E2 11258.451} C_VEL
LIN {X 0,Y 216.728,Z 681.869,A -85,B 0,C 180,E1 11257.049,E2 11257.049} C_VEL
LIN {X 0,Y 215.857,Z 680.076,A -85,B 0,C 180,E1 11256.52,E2 11256.52} C_VEL
LIN {X 0,Y 213.236,Z 677.487,A -85,B 0,C 180,E1 11255.182,E2 11255.182} C_VEL
LIN {X 0,Y 212.07,Z 674.261,A -85,B 0,C 180,E1 11254.313,E2 11254.313} C_VEL
LIN {X 0,Y 212.118,Z 674.244,A -85,B 0,C 180,E1 11248.923,E2 11248.923} C_VEL
LIN {X 0,Y 212.128,Z 674.235,A -85,B 0,C 180,E1 11243.508,E2 11243.508} C_VEL
LIN {X 0,Y 212.089,Z 674.21,A -85,B 0,C 180,E1 11238.308,E2 11238.308} C_VEL
LIN {X 0,Y 212.095,Z 674.24,A -85,B 0,C 180,E1 11232.726,E2 11232.726} C_VEL
LIN {X 0,Y 212.137,Z 674.396,A -85,B 0,C 180,E1 11229.519,E2 11229.519} C_VEL
LIN {X 0,Y 220.107,Z 694.425,A -85,B 0,C 180,E1 11224.87,E2 11224.87} C_VEL
LIN {X 0,Y 226.904,Z 713.645,A -85,B 0,C 180,E1 11220.865,E2 11220.865} C_VEL
LIN {X 0,Y 233.572,Z 735.099,A -85,B 0,C 180,E1 11216.778,E2 11216.778} C_VEL
LIN {X 0,Y 238.192,Z 752.673,A -85,B 0,C 180,E1 11213.695,E2 11213.695} C_VEL
LIN {X 0,Y 232.614,Z 795.884,A -85,B 0,C 180,E1 11208.226,E2 11208.226} C_VEL
LIN {X 0,Y 227.487,Z 839.588,A -85,B 0,C 180,E1 11202.592,E2 11202.592} C_VEL
LIN {X 0,Y 225.421,Z 855.802,A -85,B 0,C 180,E1 11200.52,E2 11200.52} C_VEL
LIN {X 0,Y 223.651,Z 867.068,A -85,B 0,C 180,E1 11199.163,E2 11199.163} C_VEL
LIN {X 0,Y 217.393,Z 984.866,A -85,B 0,C 180,E1 11193.206,E2 11193.206} C_VEL
LIN {X 0,Y 216.364,Z 1016.19,A -85,B 0,C 180,E1 11191.444,E2 11191.444} C_VEL
LIN {X 0,Y 215.394,Z 1034.197,A -85,B 0,C 180,E1 11189.928,E2 11189.928} C_VEL
LIN {X 0,Y 214.174,Z 1051.651,A -85,B 0,C 180,E1 11187.903,E2 11187.903} C_VEL
LIN {X 0,Y 212.825,Z 1068.599,A -85,B 0,C 180,E1 11185.304,E2 11185.304} C_VEL
LIN {X 0,Y 211.663,Z 1083.039,A -85,B 0,C 180,E1 11182.491,E2 11182.491} C_VEL
LIN {X 0,Y 210.759,Z 1095.941,A -85,B 0,C 180,E1 11179.389,E2 11179.389} C_VEL
LIN {X 0,Y 210.189,Z 1108.145,A -85,B 0,C 180,E1 11175.727,E2 11175.727} C_VEL
LIN {X 0,Y 210.11,Z 1117.934,A -85,B 0,C 180,E1 11172.08,E2 11172.08} C_VEL
LIN {X 0,Y 210.692,Z 1126.853,A -85,B 0,C 180,E1 11167.904,E2 11167.904} C_VEL
LIN {X 0,Y 212.104,Z 1133.63,A -85,B 0,C 180,E1 11163.778,E2 11163.778} C_VEL
LIN {X 0,Y 215.053,Z 1139.411,A -85,B 0,C 180,E1 11158.929,E2 11158.929} C_VEL
LIN {X 0,Y 219.167,Z 1142.693,A -85,B 0,C 180,E1 11154.497,E2 11154.497} C_VEL
LIN {X 0,Y 224.217,Z 1143.922,A -85,B 0,C 180,E1 11150.497,E2 11150.497} C_VEL
LIN {X 0,Y 230.781,Z 1143.297,A -85,B 0,C 180,E1 11146.464,E2 11146.464} C_VEL
LIN {X 0,Y 238,Z 1140.843,A -85,B 0,C 180,E1 11142.892,E2 11142.892} C_VEL
LIN {X 0,Y 246.134,Z 1136.513,A -85,B 0,C 180,E1 11139.547,E2 11139.547} C_VEL
LIN {X 0,Y 254.496,Z 1130.618,A -85,B 0,C 180,E1 11136.616,E2 11136.616} C_VEL
LIN {X 0,Y 263.511,Z 1122.755,A -85,B 0,C 180,E1 11133.881,E2 11133.881} C_VEL
LIN {X 0,Y 272.428,Z 1113.33,A -85,B 0,C 180,E1 11131.497,E2 11131.497} C_VEL
LIN {X 0,Y 281.081,Z 1102.482,A -85,B 0,C 180,E1 11129.419,E2 11129.419} C_VEL
LIN {X 0,Y 290.053,Z 1088.896,A -85,B 0,C 180,E1 11127.464,E2 11127.464} C_VEL
LIN {X 0,Y 297.84,Z 1074.469,A -85,B 0,C 180,E1 11125.896,E2 11125.896} C_VEL
LIN {X 0,Y 302.855,Z 1063.024,A -85,B 0,C 180,E1 11124.883,E2 11124.883} C_VEL
LIN {X 0,Y 294.765,Z 1078.647,A -85,B 0,C 180,E1 11123.666,E2 11123.666} C_VEL
LIN {X 0,Y 287.339,Z 1091.006,A -85,B 0,C 180,E1 11122.533,E2 11122.533} C_VEL
LIN {X 0,Y 282.517,Z 1098.195,A -85,B 0,C 180,E1 11122.059,E2 11122.059} C_VEL
LIN {X 0,Y 272.322,Z 1111.225,A -85,B 0,C 180,E1 11121.53,E2 11121.53} C_VEL
LIN {X 0,Y 267.589,Z 1116.719,A -85,B 0,C 180,E1 11121.008,E2 11121.008} C_VEL
LIN {X 0,Y 266.334,Z 1118.155,A -85,B 0,C 180,E1 11120.787,E2 11120.787} C_VEL
LIN {X 0,Y 254.631,Z 1130.957,A -85,B 0,C 180,E1 11118.248,E2 11118.248} C_VEL
LIN {X 0,Y 242.816,Z 1142.669,A -85,B 0,C 180,E1 11115.089,E2 11115.089} C_VEL
LIN {X 0,Y 232.202,Z 1152.418,A -85,B 0,C 180,E1 11111.535,E2 11111.535} C_VEL
LIN {X 0,Y 221.996,Z 1161.111,A -85,B 0,C 180,E1 11107.119,E2 11107.119} C_VEL
LIN {X 0,Y 214.131,Z 1167.564,A -85,B 0,C 180,E1 11102.474,E2 11102.474} C_VEL
LIN {X 0,Y 207.778,Z 1172.447,A -85,B 0,C 180,E1 11097.2,E2 11097.2} C_VEL
LIN {X 0,Y 203.768,Z 1175.504,A -85,B 0,C 180,E1 11091.589,E2 11091.589} C_VEL
LIN {X 0,Y 202.212,Z 1176.681,A -85,B 0,C 180,E1 11086.071,E2 11086.071} C_VEL
LIN {X 0,Y 201.398,Z 1185.733,A -85,B 0,C 180,E1 11080.87,E2 11080.87} C_VEL
LIN {X 0,Y 201.358,Z 1192.462,A -85,B 0,C 180,E1 11075.982,E2 11075.982} C_VEL
LIN {X 0,Y 201.447,Z 1196.876,A -85,B 0,C 180,E1 11071.987,E2 11071.987} C_VEL
LIN {X 0,Y 201.212,Z 1200.236,A -85,B 0,C 180,E1 11068.003,E2 11068.003} C_VEL
LIN {X 0,Y 200.639,Z 1203.373,A -85,B 0,C 180,E1 11062.661,E2 11062.661} C_VEL
LIN {X 0,Y 201.035,Z 1205.351,A -85,B 0,C 180,E1 11056.184,E2 11056.184} C_VEL
LIN {X 0,Y 203.928,Z 1205.918,A -85,B 0,C 180,E1 11049.023,E2 11049.023} C_VEL
LIN {X 0,Y 210.146,Z 1204.667,A -85,B 0,C 180,E1 11041.894,E2 11041.894} C_VEL
LIN {X 0,Y 221.226,Z 1201.387,A -85,B 0,C 180,E1 11034.453,E2 11034.453} C_VEL
LIN {X 0,Y 235.527,Z 1196.661,A -85,B 0,C 180,E1 11028.198,E2 11028.198} C_VEL
LIN {X 0,Y 252.57,Z 1190.52,A -85,B 0,C 180,E1 11022.921,E2 11022.921} C_VEL
LIN {X 0,Y 235.435,Z 1193.847,A -85,B 0,C 180,E1 11017.402,E2 11017.402} C_VEL
LIN {X 0,Y 221.888,Z 1195.49,A -85,B 0,C 180,E1 11011.219,E2 11011.219} C_VEL
LIN {X 0,Y 211.922,Z 1195.323,A -85,B 0,C 180,E1 11004.538,E2 11004.538} C_VEL
LIN {X 0,Y 205.394,Z 1193.499,A -85,B 0,C 180,E1 10997.573,E2 10997.573} C_VEL
LIN {X 0,Y 201.946,Z 1190.251,A -85,B 0,C 180,E1 10990.851,E2 10990.851} C_VEL
LIN {X 0,Y 200.626,Z 1185.899,A -85,B 0,C 180,E1 10984.866,E2 10984.866} C_VEL
LIN {X 0,Y 200.296,Z 1180.73,A -85,B 0,C 180,E1 10979.434,E2 10979.434} C_VEL
LIN {X 0,Y 200.363,Z 1174.366,A -85,B 0,C 180,E1 10974.278,E2 10974.278} C_VEL
LIN {X 0,Y 200.958,Z 1166.118,A -85,B 0,C 180,E1 10968.817,E2 10968.817} C_VEL
LIN {X 0,Y 202.349,Z 1156.492,A -85,B 0,C 180,E1 10963.647,E2 10963.647} C_VEL
LIN {X 0,Y 204.916,Z 1144.335,A -85,B 0,C 180,E1 10958.239,E2 10958.239} C_VEL
LIN {X 0,Y 208.52,Z 1130.642,A -85,B 0,C 180,E1 10953.216,E2 10953.216} C_VEL
LIN {X 0,Y 213.005,Z 1115.489,A -85,B 0,C 180,E1 10948.604,E2 10948.604} C_VEL
LIN {X 0,Y 218.208,Z 1098.802,A -85,B 0,C 180,E1 10944.42,E2 10944.42} C_VEL
LIN {X 0,Y 223.917,Z 1080.566,A -85,B 0,C 180,E1 10940.655,E2 10940.655} C_VEL
LIN {X 0,Y 229.951,Z 1060.79,A -85,B 0,C 180,E1 10937.295,E2 10937.295} C_VEL
LIN {X 0,Y 236.138,Z 1039.321,A -85,B 0,C 180,E1 10934.316,E2 10934.316} C_VEL
LIN {X 0,Y 242.183,Z 1016.355,A -85,B 0,C 180,E1 10931.754,E2 10931.754} C_VEL
LIN {X 0,Y 247.86,Z 992.008,A -85,B 0,C 180,E1 10929.6,E2 10929.6} C_VEL
LIN {X 0,Y 252.685,Z 967.655,A -85,B 0,C 180,E1 10927.916,E2 10927.916} C_VEL
LIN {X 0,Y 256.871,Z 941.964,A -85,B 0,C 180,E1 10926.578,E2 10926.578} C_VEL
LIN {X 0,Y 276.958,Z 795.481,A -85,B 0,C 180,E1 10921.025,E2 10921.025} C_VEL
LIN {X 0,Y 263.52,Z 769.994,A -85,B 0,C 180,E1 10917.027,E2 10917.027} C_VEL
LIN {X 0,Y 251.272,Z 748.033,A -85,B 0,C 180,E1 10912.956,E2 10912.956} C_VEL
LIN {X 0,Y 240.681,Z 730.087,A -85,B 0,C 180,E1 10909.037,E2 10909.037} C_VEL
LIN {X 0,Y 229.49,Z 712.26,A -85,B 0,C 180,E1 10904.383,E2 10904.383} C_VEL
LIN {X 0,Y 221.988,Z 701.228,A -85,B 0,C 180,E1 10900.946,E2 10900.946} C_VEL
LIN {X 0,Y 218.49,Z 696.197,A -85,B 0,C 180,E1 10899.22,E2 10899.22} C_VEL
LIN {X 0,Y 215.489,Z 691.836,A -85,B 0,C 180,E1 10897.67,E2 10897.67} C_VEL
LIN {X 0,Y 212.558,Z 687.651,A -85,B 0,C 180,E1 10896.079,E2 10896.079} C_VEL
LIN {X 0,Y 209.012,Z 683.002,A -85,B 0,C 180,E1 10894.05,E2 10894.05} C_VEL
LIN {X 0,Y 208.121,Z 681.186,A -85,B 0,C 180,E1 10893.447,E2 10893.447} C_VEL
LIN {X 0,Y 205.439,Z 678.707,A -85,B 0,C 180,E1 10891.956,E2 10891.956} C_VEL
LIN {X 0,Y 204.199,Z 675.519,A -85,B 0,C 180,E1 10890.986,E2 10890.986} C_VEL
LIN {X 0,Y 204.157,Z 675.219,A -85,B 0,C 180,E1 10890.846,E2 10890.846} C_VEL
LIN {X 0,Y 204.184,Z 675.201,A -85,B 0,C 180,E1 10885.229,E2 10885.229} C_VEL
LIN {X 0,Y 204.167,Z 675.203,A -85,B 0,C 180,E1 10880.134,E2 10880.134} C_VEL
LIN {X 0,Y 204.148,Z 675.237,A -85,B 0,C 180,E1 10874.377,E2 10874.377} C_VEL
LIN {X 0,Y 204.201,Z 675.439,A -85,B 0,C 180,E1 10870.927,E2 10870.927} C_VEL
LIN {X 0,Y 211.777,Z 694.081,A -85,B 0,C 180,E1 10866.344,E2 10866.344} C_VEL
LIN {X 0,Y 218.577,Z 713.034,A -85,B 0,C 180,E1 10862.191,E2 10862.191} C_VEL
LIN {X 0,Y 224.925,Z 733.028,A -85,B 0,C 180,E1 10858.216,E2 10858.216} C_VEL
LIN {X 0,Y 230.717,Z 754.312,A -85,B 0,C 180,E1 10854.35,E2 10854.35} C_VEL
LIN {X 0,Y 225.108,Z 796.45,A -85,B 0,C 180,E1 10848.904,E2 10848.904} C_VEL
LIN {X 0,Y 219.706,Z 840.963,A -85,B 0,C 180,E1 10843.043,E2 10843.043} C_VEL
LIN {X 0,Y 217.863,Z 855.086,A -85,B 0,C 180,E1 10841.183,E2 10841.183} C_VEL
LIN {X 0,Y 215.779,Z 868.047,A -85,B 0,C 180,E1 10839.571,E2 10839.571} C_VEL
LIN {X 0,Y 209.433,Z 984.558,A -85,B 0,C 180,E1 10833.412,E2 10833.412} C_VEL
LIN {X 0,Y 208.333,Z 1017.001,A -85,B 0,C 180,E1 10831.505,E2 10831.505} C_VEL
LIN {X 0,Y 207.347,Z 1034.916,A -85,B 0,C 180,E1 10829.933,E2 10829.933} C_VEL
LIN {X 0,Y 206.063,Z 1052.896,A -85,B 0,C 180,E1 10827.756,E2 10827.756} C_VEL
LIN {X 0,Y 204.741,Z 1069.344,A -85,B 0,C 180,E1 10825.136,E2 10825.136} C_VEL
LIN {X 0,Y 203.583,Z 1083.754,A -85,B 0,C 180,E1 10822.214,E2 10822.214} C_VEL
LIN {X 0,Y 202.705,Z 1096.659,A -85,B 0,C 180,E1 10818.993,E2 10818.993} C_VEL
LIN {X 0,Y 202.178,Z 1108.897,A -85,B 0,C 180,E1 10815.189,E2 10815.189} C_VEL
LIN {X 0,Y 202.176,Z 1118.704,A -85,B 0,C 180,E1 10811.403,E2 10811.403} C_VEL
LIN {X 0,Y 202.891,Z 1127.673,A -85,B 0,C 180,E1 10807.071,E2 10807.071} C_VEL
LIN {X 0,Y 204.504,Z 1134.534,A -85,B 0,C 180,E1 10802.796,E2 10802.796} C_VEL
LIN {X 0,Y 207.562,Z 1140.164,A -85,B 0,C 180,E1 10798.062,E2 10798.062} C_VEL
LIN {X 0,Y 211.681,Z 1143.499,A -85,B 0,C 180,E1 10793.757,E2 10793.757} C_VEL
LIN {X 0,Y 217.372,Z 1145.153,A -85,B 0,C 180,E1 10789.392,E2 10789.392} C_VEL
LIN {X 0,Y 223.89,Z 1144.837,A -85,B 0,C 180,E1 10785.511,E2 10785.511} C_VEL
LIN {X 0,Y 231.457,Z 1142.786,A -85,B 0,C 180,E1 10781.873,E2 10781.873} C_VEL
LIN {X 0,Y 239.408,Z 1139.196,A -85,B 0,C 180,E1 10778.688,E2 10778.688} C_VEL
LIN {X 0,Y 248.685,Z 1133.437,A -85,B 0,C 180,E1 10775.53,E2 10775.53} C_VEL
LIN {X 0,Y 258.073,Z 1126.087,A -85,B 0,C 180,E1 10772.79,E2 10772.79} C_VEL
LIN {X 0,Y 268.031,Z 1116.555,A -85,B 0,C 180,E1 10770.249,E2 10770.249} C_VEL
LIN {X 0,Y 277.729,Z 1105.255,A -85,B 0,C 180,E1 10768.042,E2 10768.042} C_VEL
LIN {X 0,Y 286.354,Z 1093.234,A -85,B 0,C 180,E1 10766.271,E2 10766.271} C_VEL
LIN {X 0,Y 292.879,Z 1082.463,A -85,B 0,C 180,E1 10765.015,E2 10765.015} C_VEL
LIN {X 0,Y 282.217,Z 1098.243,A -85,B 0,C 180,E1 10763.532,E2 10763.532} C_VEL
LIN {X 0,Y 270.517,Z 1113.224,A -85,B 0,C 180,E1 10761.585,E2 10761.585} C_VEL
LIN {X 0,Y 266.334,Z 1118.155,A -85,B 0,C 180,E1 10760.787,E2 10760.787} C_VEL
LIN {X 0,Y 261.507,Z 1123.386,A -85,B 0,C 180,E1 10760.083,E2 10760.083} C_VEL
LIN {X 0,Y 248.883,Z 1134.882,A -85,B 0,C 180,E1 10758.886,E2 10758.886} C_VEL
LIN {X 0,Y 243.649,Z 1139.269,A -85,B 0,C 180,E1 10758.067,E2 10758.067} C_VEL
LIN {X 0,Y 242.322,Z 1140.394,A -85,B 0,C 180,E1 10757.757,E2 10757.757} C_VEL
LIN {X 0,Y 230.267,Z 1150.536,A -85,B 0,C 180,E1 10754.229,E2 10754.229} C_VEL
LIN {X 0,Y 219.169,Z 1159.057,A -85,B 0,C 180,E1 10750.03,E2 10750.03} C_VEL
LIN {X 0,Y 209.714,Z 1165.85,A -85,B 0,C 180,E1 10745.228,E2 10745.228} C_VEL
LIN {X 0,Y 202.326,Z 1170.745,A -85,B 0,C 180,E1 10739.938,E2 10739.938} C_VEL
LIN {X 0,Y 197.081,Z 1173.947,A -85,B 0,C 180,E1 10734.032,E2 10734.032} C_VEL
LIN {X 0,Y 194.618,Z 1175.126,A -85,B 0,C 180,E1 10728.26,E2 10728.26} C_VEL
LIN {X 0,Y 194.363,Z 1175.152,A -85,B 0,C 180,E1 10726.278,E2 10726.278} C_VEL
LIN {X 0,Y 193.526,Z 1184.129,A -85,B 0,C 180,E1 10720.959,E2 10720.959} C_VEL
LIN {X 0,Y 193.491,Z 1191.38,A -85,B 0,C 180,E1 10715.63,E2 10715.63} C_VEL
LIN {X 0,Y 193.583,Z 1195.824,A -85,B 0,C 180,E1 10711.476,E2 10711.476} C_VEL
LIN {X 0,Y 193.308,Z 1199,A -85,B 0,C 180,E1 10707.624,E2 10707.624} C_VEL
LIN {X 0,Y 192.785,Z 1201.83,A -85,B 0,C 180,E1 10702.845,E2 10702.845} C_VEL
LIN {X 0,Y 193.083,Z 1204.281,A -85,B 0,C 180,E1 10696.215,E2 10696.215} C_VEL
LIN {X 0,Y 196.002,Z 1205.173,A -85,B 0,C 180,E1 10688.761,E2 10688.761} C_VEL
LIN {X 0,Y 203.001,Z 1204.349,A -85,B 0,C 180,E1 10680.811,E2 10680.811} C_VEL
LIN {X 0,Y 213.482,Z 1201.879,A -85,B 0,C 180,E1 10673.829,E2 10673.829} C_VEL
LIN {X 0,Y 228.436,Z 1197.586,A -85,B 0,C 180,E1 10667.273,E2 10667.273} C_VEL
LIN {X 0,Y 242.396,Z 1193.262,A -85,B 0,C 180,E1 10662.899,E2 10662.899} C_VEL
LIN {X 0,Y 225.388,Z 1195.683,A -85,B 0,C 180,E1 10657.115,E2 10657.115} C_VEL
LIN {X 0,Y 212.07,Z 1196.365,A -85,B 0,C 180,E1 10650.617,E2 10650.617} C_VEL
LIN {X 0,Y 202.473,Z 1195.342,A -85,B 0,C 180,E1 10643.585,E2 10643.585} C_VEL
LIN {X 0,Y 196.244,Z 1192.548,A -85,B 0,C 180,E1 10635.976,E2 10635.976} C_VEL
LIN {X 0,Y 193.361,Z 1188.431,A -85,B 0,C 180,E1 10628.931,E2 10628.931} C_VEL
LIN {X 0,Y 192.456,Z 1183.22,A -85,B 0,C 180,E1 10622.686,E2 10622.686} C_VEL
LIN {X 0,Y 192.307,Z 1177.551,A -85,B 0,C 180,E1 10617.324,E2 10617.324} C_VEL
LIN {X 0,Y 192.566,Z 1170.344,A -85,B 0,C 180,E1 10611.947,E2 10611.947} C_VEL
LIN {X 0,Y 193.459,Z 1161.647,A -85,B 0,C 180,E1 10606.558,E2 10606.558} C_VEL
LIN {X 0,Y 195.32,Z 1151.068,A -85,B 0,C 180,E1 10601.192,E2 10601.192} C_VEL
LIN {X 0,Y 198.515,Z 1137.786,A -85,B 0,C 180,E1 10595.613,E2 10595.613} C_VEL
LIN {X 0,Y 202.521,Z 1123.804,A -85,B 0,C 180,E1 10590.747,E2 10590.747} C_VEL
LIN {X 0,Y 207.634,Z 1107.414,A -85,B 0,C 180,E1 10586.048,E2 10586.048} C_VEL
LIN {X 0,Y 213.643,Z 1088.75,A -85,B 0,C 180,E1 10581.683,E2 10581.683} C_VEL
LIN {X 0,Y 219.865,Z 1069.16,A -85,B 0,C 180,E1 10577.957,E2 10577.957} C_VEL
LIN {X 0,Y 226.048,Z 1048.753,A -85,B 0,C 180,E1 10574.8,E2 10574.8} C_VEL
LIN {X 0,Y 232.218,Z 1026.836,A -85,B 0,C 180,E1 10572.043,E2 10572.043} C_VEL
LIN {X 0,Y 237.973,Z 1004.211,A -85,B 0,C 180,E1 10569.754,E2 10569.754} C_VEL
LIN {X 0,Y 243.339,Z 980.071,A -85,B 0,C 180,E1 10567.818,E2 10567.818} C_VEL
LIN {X 0,Y 248.069,Z 954.6,A -85,B 0,C 180,E1 10566.253,E2 10566.253} C_VEL
LIN {X 0,Y 252.853,Z 921.826,A -85,B 0,C 180,E1 10564.79,E2 10564.79} C_VEL
LIN {X 0,Y 270.353,Z 798.201,A -85,B 0,C 180,E1 10560.056,E2 10560.056} C_VEL
LIN {X 0,Y 257.013,Z 772.847,A -85,B 0,C 180,E1 10555.927,E2 10555.927} C_VEL
LIN {X 0,Y 245.066,Z 751.189,A -85,B 0,C 180,E1 10551.767,E2 10551.767} C_VEL
LIN {X 0,Y 234.561,Z 733.544,A -85,B 0,C 180,E1 10547.717,E2 10547.717} C_VEL
LIN {X 0,Y 224.857,Z 717.922,A -85,B 0,C 180,E1 10543.504,E2 10543.504} C_VEL
LIN {X 0,Y 217.759,Z 707.276,A -85,B 0,C 180,E1 10540.119,E2 10540.119} C_VEL
LIN {X 0,Y 211.884,Z 698.607,A -85,B 0,C 180,E1 10537.051,E2 10537.051} C_VEL
LIN {X 0,Y 208.632,Z 693.829,A -85,B 0,C 180,E1 10535.194,E2 10535.194} C_VEL
LIN {X 0,Y 205.335,Z 689.57,A -85,B 0,C 180,E1 10533.277,E2 10533.277} C_VEL
LIN {X 0,Y 204.38,Z 687.975,A -85,B 0,C 180,E1 10532.654,E2 10532.654} C_VEL
LIN {X 0,Y 201.489,Z 684.699,A -85,B 0,C 180,E1 10530.928,E2 10530.928} C_VEL
LIN {X 0,Y 200.259,Z 682.224,A -85,B 0,C 180,E1 10530.004,E2 10530.004} C_VEL
LIN {X 0,Y 197.454,Z 679.575,A -85,B 0,C 180,E1 10528.19,E2 10528.19} C_VEL
LIN {X 0,Y 196.275,Z 676.458,A -85,B 0,C 180,E1 10527.084,E2 10527.084} C_VEL
LIN {X 0,Y 196.237,Z 676.188,A -85,B 0,C 180,E1 10526.206,E2 10526.206} C_VEL
LIN {X 0,Y 196.237,Z 676.196,A -85,B 0,C 180,E1 10520.62,E2 10520.62} C_VEL
LIN {X 0,Y 196.209,Z 676.228,A -85,B 0,C 180,E1 10514.638,E2 10514.638} C_VEL
LIN {X 0,Y 196.237,Z 676.336,A -85,B 0,C 180,E1 10512.433,E2 10512.433} C_VEL
LIN {X 0,Y 197.247,Z 679.258,A -85,B 0,C 180,E1 10511.686,E2 10511.686} C_VEL
LIN {X 0,Y 203.023,Z 692.716,A -85,B 0,C 180,E1 10508.176,E2 10508.176} C_VEL
LIN {X 0,Y 209.524,Z 710.16,A -85,B 0,C 180,E1 10504.114,E2 10504.114} C_VEL
LIN {X 0,Y 216.266,Z 730.966,A -85,B 0,C 180,E1 10499.743,E2 10499.743} C_VEL
LIN {X 0,Y 221.95,Z 751.157,A -85,B 0,C 180,E1 10495.889,E2 10495.889} C_VEL
LIN {X 0,Y 223.19,Z 756.443,A -85,B 0,C 180,E1 10494.936,E2 10494.936} C_VEL
LIN {X 0,Y 217.157,Z 800.128,A -85,B 0,C 180,E1 10489.175,E2 10489.175} C_VEL
LIN {X 0,Y 211.655,Z 844.125,A -85,B 0,C 180,E1 10483.227,E2 10483.227} C_VEL
LIN {X 0,Y 209.923,Z 856.249,A -85,B 0,C 180,E1 10481.606,E2 10481.606} C_VEL
LIN {X 0,Y 207.898,Z 868.964,A -85,B 0,C 180,E1 10479.985,E2 10479.985} C_VEL
LIN {X 0,Y 201.459,Z 984.494,A -85,B 0,C 180,E1 10473.592,E2 10473.592} C_VEL
LIN {X 0,Y 200.292,Z 1017.934,A -85,B 0,C 180,E1 10471.542,E2 10471.542} C_VEL
LIN {X 0,Y 199.303,Z 1035.521,A -85,B 0,C 180,E1 10469.938,E2 10469.938} C_VEL
LIN {X 0,Y 198,Z 1053.446,A -85,B 0,C 180,E1 10467.676,E2 10467.676} C_VEL
LIN {X 0,Y 196.672,Z 1069.873,A -85,B 0,C 180,E1 10464.952,E2 10464.952} C_VEL
LIN {X 0,Y 195.513,Z 1084.38,A -85,B 0,C 180,E1 10461.914,E2 10461.914} C_VEL
LIN {X 0,Y 194.634,Z 1097.811,A -85,B 0,C 180,E1 10458.411,E2 10458.411} C_VEL
LIN {X 0,Y 194.169,Z 1110.407,A -85,B 0,C 180,E1 10454.304,E2 10454.304} C_VEL
LIN {X 0,Y 194.299,Z 1120.08,A -85,B 0,C 180,E1 10450.37,E2 10450.37} C_VEL
LIN {X 0,Y 195.22,Z 1128.981,A -85,B 0,C 180,E1 10445.873,E2 10445.873} C_VEL
LIN {X 0,Y 197.128,Z 1135.775,A -85,B 0,C 180,E1 10441.447,E2 10441.447} C_VEL
LIN {X 0,Y 200.849,Z 1141.653,A -85,B 0,C 180,E1 10436.283,E2 10436.283} C_VEL
LIN {X 0,Y 205.843,Z 1145.047,A -85,B 0,C 180,E1 10431.615,E2 10431.615} C_VEL
LIN {X 0,Y 211.82,Z 1146.46,A -85,B 0,C 180,E1 10427.453,E2 10427.453} C_VEL
LIN {X 0,Y 219.421,Z 1146.003,A -85,B 0,C 180,E1 10423.311,E2 10423.311} C_VEL
LIN {X 0,Y 227.662,Z 1143.811,A -85,B 0,C 180,E1 10419.693,E2 10419.693} C_VEL
LIN {X 0,Y 236.924,Z 1139.669,A -85,B 0,C 180,E1 10416.31,E2 10416.31} C_VEL
LIN {X 0,Y 246.146,Z 1134.169,A -85,B 0,C 180,E1 10413.454,E2 10413.454} C_VEL
LIN {X 0,Y 256.783,Z 1126.064,A -85,B 0,C 180,E1 10410.613,E2 10410.613} C_VEL
LIN {X 0,Y 266.839,Z 1116.684,A -85,B 0,C 180,E1 10408.27,E2 10408.27} C_VEL
LIN {X 0,Y 276.817,Z 1105.486,A -85,B 0,C 180,E1 10406.198,E2 10406.198} C_VEL
LIN {X 0,Y 281.742,Z 1099.017,A -85,B 0,C 180,E1 10405.215,E2 10405.215} C_VEL
LIN {X 0,Y 269.994,Z 1113.085,A -85,B 0,C 180,E1 10403.472,E2 10403.472} C_VEL
LIN {X 0,Y 257.673,Z 1126.056,A -85,B 0,C 180,E1 10401.252,E2 10401.252} C_VEL
LIN {X 0,Y 245.459,Z 1137.656,A -85,B 0,C 180,E1 10398.544,E2 10398.544} C_VEL
LIN {X 0,Y 242.322,Z 1140.394,A -85,B 0,C 180,E1 10397.757,E2 10397.757} C_VEL
LIN {X 0,Y 237.213,Z 1144.474,A -85,B 0,C 180,E1 10396.728,E2 10396.728} C_VEL
LIN {X 0,Y 223.775,Z 1153.039,A -85,B 0,C 180,E1 10394.715,E2 10394.715} C_VEL
LIN {X 0,Y 218.515,Z 1156.157,A -85,B 0,C 180,E1 10393.502,E2 10393.502} C_VEL
LIN {X 0,Y 217.257,Z 1156.948,A -85,B 0,C 180,E1 10393.078,E2 10393.078} C_VEL
LIN {X 0,Y 206.381,Z 1163.903,A -85,B 0,C 180,E1 10388.321,E2 10388.321} C_VEL
LIN {X 0,Y 197.817,Z 1168.878,A -85,B 0,C 180,E1 10383.081,E2 10383.081} C_VEL
LIN {X 0,Y 191.434,Z 1172.099,A -85,B 0,C 180,E1 10377.359,E2 10377.359} C_VEL
LIN {X 0,Y 187.614,Z 1173.584,A -85,B 0,C 180,E1 10371.243,E2 10371.243} C_VEL
LIN {X 0,Y 186.539,Z 1173.529,A -85,B 0,C 180,E1 10366.5,E2 10366.5} C_VEL
LIN {X 0,Y 185.647,Z 1182.772,A -85,B 0,C 180,E1 10360.861,E2 10360.861} C_VEL
LIN {X 0,Y 185.638,Z 1190.254,A -85,B 0,C 180,E1 10355.249,E2 10355.249} C_VEL
LIN {X 0,Y 185.72,Z 1195.001,A -85,B 0,C 180,E1 10350.613,E2 10350.613} C_VEL
LIN {X 0,Y 185.297,Z 1198.334,A -85,B 0,C 180,E1 10346.283,E2 10346.283} C_VEL
LIN {X 0,Y 184.828,Z 1201.359,A -85,B 0,C 180,E1 10340.656,E2 10340.656} C_VEL
LIN {X 0,Y 186.061,Z 1203.784,A -85,B 0,C 180,E1 10332.804,E2 10332.804} C_VEL
LIN {X 0,Y 190.409,Z 1204.442,A -85,B 0,C 180,E1 10325.155,E2 10325.155} C_VEL
LIN {X 0,Y 199.608,Z 1203.325,A -85,B 0,C 180,E1 10316.902,E2 10316.902} C_VEL
LIN {X 0,Y 213.007,Z 1200.528,A -85,B 0,C 180,E1 10309.62,E2 10309.62} C_VEL
LIN {X 0,Y 230.044,Z 1196.104,A -85,B 0,C 180,E1 10303.455,E2 10303.455} C_VEL
LIN {X 0,Y 232.056,Z 1195.562,A -85,B 0,C 180,E1 10302.836,E2 10302.836} C_VEL
LIN {X 0,Y 215.329,Z 1197.055,A -85,B 0,C 180,E1 10296.806,E2 10296.806} C_VEL
LIN {X 0,Y 202.259,Z 1196.812,A -85,B 0,C 180,E1 10289.96,E2 10289.96} C_VEL
LIN {X 0,Y 192.796,Z 1194.842,A -85,B 0,C 180,E1 10282.253,E2 10282.253} C_VEL
LIN {X 0,Y 187.515,Z 1191.479,A -85,B 0,C 180,E1 10274.836,E2 10274.836} C_VEL
LIN {X 0,Y 185.118,Z 1186.758,A -85,B 0,C 180,E1 10267.767,E2 10267.767} C_VEL
LIN {X 0,Y 184.423,Z 1180.964,A -85,B 0,C 180,E1 10261.249,E2 10261.249} C_VEL
LIN {X 0,Y 184.37,Z 1174.973,A -85,B 0,C 180,E1 10255.964,E2 10255.964} C_VEL
LIN {X 0,Y 184.775,Z 1167.24,A -85,B 0,C 180,E1 10250.35,E2 10250.35} C_VEL
LIN {X 0,Y 185.982,Z 1157.74,A -85,B 0,C 180,E1 10244.733,E2 10244.733} C_VEL
LIN {X 0,Y 188.425,Z 1145.729,A -85,B 0,C 180,E1 10238.855,E2 10238.855} C_VEL
LIN {X 0,Y 192.008,Z 1132.242,A -85,B 0,C 180,E1 10233.402,E2 10233.402} C_VEL
LIN {X 0,Y 196.569,Z 1117.256,A -85,B 0,C 180,E1 10228.412,E2 10228.412} C_VEL
LIN {X 0,Y 202.147,Z 1100.098,A -85,B 0,C 180,E1 10223.737,E2 10223.737} C_VEL
LIN {X 0,Y 208.044,Z 1082.167,A -85,B 0,C 180,E1 10219.736,E2 10219.736} C_VEL
LIN {X 0,Y 214.344,Z 1062.605,A -85,B 0,C 180,E1 10216.162,E2 10216.162} C_VEL
LIN {X 0,Y 221.063,Z 1040.525,A -85,B 0,C 180,E1 10212.893,E2 10212.893} C_VEL
LIN {X 0,Y 227.547,Z 1017.255,A -85,B 0,C 180,E1 10210.139,E2 10210.139} C_VEL
LIN {X 0,Y 233.499,Z 993.107,A -85,B 0,C 180,E1 10207.889,E2 10207.889} C_VEL
LIN {X 0,Y 238.739,Z 968.11,A -85,B 0,C 180,E1 10206.078,E2 10206.078} C_VEL
LIN {X 0,Y 243.204,Z 942.111,A -85,B 0,C 180,E1 10204.667,E2 10204.667} C_VEL
LIN {X 0,Y 263.734,Z 800.992,A -85,B 0,C 180,E1 10199.065,E2 10199.065} C_VEL
LIN {X 0,Y 251.371,Z 777.226,A -85,B 0,C 180,E1 10195.067,E2 10195.067} C_VEL
LIN {X 0,Y 239.774,Z 756.046,A -85,B 0,C 180,E1 10190.891,E2 10190.891} C_VEL
LIN {X 0,Y 229.728,Z 738.93,A -85,B 0,C 180,E1 10186.86,E2 10186.86} C_VEL
LIN {X 0,Y 220.238,Z 723.521,A -85,B 0,C 180,E1 10182.581,E2 10182.581} C_VEL
LIN {X 0,Y 213.516,Z 713.245,A -85,B 0,C 180,E1 10179.24,E2 10179.24} C_VEL
LIN {X 0,Y 207.694,Z 704.675,A -85,B 0,C 180,E1 10176.083,E2 10176.083} C_VEL
LIN {X 0,Y 204.011,Z 699.482,A -85,B 0,C 180,E1 10173.938,E2 10173.938} C_VEL
LIN {X 0,Y 200.553,Z 694.574,A -85,B 0,C 180,E1 10171.79,E2 10171.79} C_VEL
LIN {X 0,Y 197.613,Z 690.662,A -85,B 0,C 180,E1 10169.859,E2 10169.859} C_VEL
LIN {X 0,Y 196.625,Z 689.057,A -85,B 0,C 180,E1 10169.13,E2 10169.13} C_VEL
LIN {X 0,Y 193.755,Z 685.731,A -85,B 0,C 180,E1 10167.12,E2 10167.12} C_VEL
LIN {X 0,Y 192.631,Z 683.33,A -85,B 0,C 180,E1 10166.135,E2 10166.135} C_VEL
LIN {X 0,Y 189.675,Z 680.759,A -85,B 0,C 180,E1 10164.036,E2 10164.036} C_VEL
LIN {X 0,Y 188.41,Z 677.751,A -85,B 0,C 180,E1 10162.737,E2 10162.737} C_VEL
LIN {X 0,Y 188.322,Z 677.211,A -85,B 0,C 180,E1 10162.53,E2 10162.53} C_VEL
LIN {X 0,Y 188.265,Z 677.192,A -85,B 0,C 180,E1 10156.49,E2 10156.49} C_VEL
LIN {X 0,Y 188.274,Z 677.307,A -85,B 0,C 180,E1 10154.052,E2 10154.052} C_VEL
LIN {X 0,Y 189.549,Z 680.66,A -85,B 0,C 180,E1 10153.139,E2 10153.139} C_VEL
LIN {X 0,Y 195.9,Z 695.522,A -85,B 0,C 180,E1 10149.071,E2 10149.071} C_VEL
LIN {X 0,Y 202.165,Z 712.397,A -85,B 0,C 180,E1 10144.988,E2 10144.988} C_VEL
LIN {X 0,Y 208.751,Z 732.632,A -85,B 0,C 180,E1 10140.601,E2 10140.601} C_VEL
LIN {X 0,Y 214.581,Z 753.423,A -85,B 0,C 180,E1 10136.509,E2 10136.509} C_VEL
LIN {X 0,Y 215.657,Z 758.767,A -85,B 0,C 180,E1 10135.558,E2 10135.558} C_VEL
LIN {X 0,Y 209.516,Z 801.63,A -85,B 0,C 180,E1 10129.77,E2 10129.77} C_VEL
LIN {X 0,Y 203.743,Z 846.312,A -85,B 0,C 180,E1 10123.582,E2 10123.582} C_VEL
LIN {X 0,Y 201.859,Z 858.161,A -85,B 0,C 180,E1 10121.958,E2 10121.958} C_VEL
LIN {X 0,Y 200.018,Z 869.849,A -85,B 0,C 180,E1 10120.416,E2 10120.416} C_VEL
LIN {X 0,Y 193.511,Z 983.516,A -85,B 0,C 180,E1 10113.823,E2 10113.823} C_VEL
LIN {X 0,Y 192.258,Z 1018.596,A -85,B 0,C 180,E1 10111.569,E2 10111.569} C_VEL
LIN {X 0,Y 191.226,Z 1036.491,A -85,B 0,C 180,E1 10109.863,E2 10109.863} C_VEL
LIN {X 0,Y 189.945,Z 1053.845,A -85,B 0,C 180,E1 10107.588,E2 10107.588} C_VEL
LIN {X 0,Y 188.676,Z 1069.499,A -85,B 0,C 180,E1 10104.91,E2 10104.91} C_VEL
LIN {X 0,Y 187.507,Z 1084.203,A -85,B 0,C 180,E1 10101.746,E2 10101.746} C_VEL
LIN {X 0,Y 186.605,Z 1098.372,A -85,B 0,C 180,E1 10097.938,E2 10097.938} C_VEL
LIN {X 0,Y 186.215,Z 1110.112,A -85,B 0,C 180,E1 10093.976,E2 10093.976} C_VEL
LIN {X 0,Y 186.384,Z 1120.077,A -85,B 0,C 180,E1 10089.878,E2 10089.878} C_VEL
LIN {X 0,Y 187.42,Z 1129.126,A -85,B 0,C 180,E1 10085.197,E2 10085.197} C_VEL
LIN {X 0,Y 189.5,Z 1136.209,A -85,B 0,C 180,E1 10080.598,E2 10080.598} C_VEL
LIN {X 0,Y 192.987,Z 1141.687,A -85,B 0,C 180,E1 10075.834,E2 10075.834} C_VEL
LIN {X 0,Y 197.816,Z 1145.497,A -85,B 0,C 180,E1 10071.272,E2 10071.272} C_VEL
LIN {X 0,Y 203.936,Z 1147.46,A -85,B 0,C 180,E1 10066.96,E2 10066.96} C_VEL
LIN {X 0,Y 211.761,Z 1147.679,A -85,B 0,C 180,E1 10062.688,E2 10062.688} C_VEL
LIN {X 0,Y 220.242,Z 1146.09,A -85,B 0,C 180,E1 10058.977,E2 10058.977} C_VEL
LIN {X 0,Y 230.302,Z 1142.445,A -85,B 0,C 180,E1 10055.362,E2 10055.362} C_VEL
LIN {X 0,Y 240.619,Z 1137.032,A -85,B 0,C 180,E1 10052.258,E2 10052.258} C_VEL
LIN {X 0,Y 251.678,Z 1129.554,A -85,B 0,C 180,E1 10049.429,E2 10049.429} C_VEL
LIN {X 0,Y 262.592,Z 1120.301,A -85,B 0,C 180,E1 10047.004,E2 10047.004} C_VEL
LIN {X 0,Y 270.329,Z 1112.526,A -85,B 0,C 180,E1 10045.417,E2 10045.417} C_VEL
LIN {X 0,Y 258.497,Z 1124.271,A -85,B 0,C 180,E1 10043.562,E2 10043.562} C_VEL
LIN {X 0,Y 245.524,Z 1135.816,A -85,B 0,C 180,E1 10041.057,E2 10041.057} C_VEL
LIN {X 0,Y 232.098,Z 1146.433,A -85,B 0,C 180,E1 10037.809,E2 10037.809} C_VEL
LIN {X 0,Y 219.974,Z 1155.133,A -85,B 0,C 180,E1 10034.058,E2 10034.058} C_VEL
LIN {X 0,Y 217.257,Z 1156.948,A -85,B 0,C 180,E1 10033.078,E2 10033.078} C_VEL
LIN {X 0,Y 212.385,Z 1159.72,A -85,B 0,C 180,E1 10031.629,E2 10031.629} C_VEL
LIN {X 0,Y 199.438,Z 1164.968,A -85,B 0,C 180,E1 10028.523,E2 10028.523} C_VEL
LIN {X 0,Y 194.494,Z 1166.804,A -85,B 0,C 180,E1 10026.668,E2 10026.668} C_VEL
LIN {X 0,Y 193.749,Z 1167.122,A -85,B 0,C 180,E1 10026.243,E2 10026.243} C_VEL
LIN {X 0,Y 185.663,Z 1170.581,A -85,B 0,C 180,E1 10020.051,E2 10020.051} C_VEL
LIN {X 0,Y 180.842,Z 1172.045,A -85,B 0,C 180,E1 10013.8,E2 10013.8} C_VEL
LIN {X 0,Y 178.845,Z 1171.737,A -85,B 0,C 180,E1 10007.567,E2 10007.567} C_VEL
LIN {X 0,Y 178.749,Z 1171.769,A -85,B 0,C 180,E1 10006.738,E2 10006.738} C_VEL
LIN {X 0,Y 177.773,Z 1181.462,A -85,B 0,C 180,E1 10000.692,E2 10000.692} C_VEL
LIN {X 0,Y 177.794,Z 1188.662,A -85,B 0,C 180,E1 9995.158,E2 9995.158} C_VEL
LIN {X 0,Y 177.876,Z 1193.599,A -85,B 0,C 180,E1 9990.318,E2 9990.318} C_VEL
LIN {X 0,Y 177.361,Z 1197.216,A -85,B 0,C 180,E1 9985.469,E2 9985.469} C_VEL
LIN {X 0,Y 176.984,Z 1200.405,A -85,B 0,C 180,E1 9979.251,E2 9979.251} C_VEL
LIN {X 0,Y 178.619,Z 1202.864,A -85,B 0,C 180,E1 9971.388,E2 9971.388} C_VEL
LIN {X 0,Y 183.991,Z 1203.661,A -85,B 0,C 180,E1 9963.043,E2 9963.043} C_VEL
LIN {X 0,Y 194.114,Z 1202.813,A -85,B 0,C 180,E1 9954.762,E2 9954.762} C_VEL
LIN {X 0,Y 208.018,Z 1200.345,A -85,B 0,C 180,E1 9947.701,E2 9947.701} C_VEL
LIN {X 0,Y 221.686,Z 1197.391,A -85,B 0,C 180,E1 9942.765,E2 9942.765} C_VEL
LIN {X 0,Y 205.261,Z 1197.931,A -85,B 0,C 180,E1 9936.469,E2 9936.469} C_VEL
LIN {X 0,Y 192.42,Z 1196.819,A -85,B 0,C 180,E1 9929.185,E2 9929.185} C_VEL
LIN {X 0,Y 183.483,Z 1193.995,A -85,B 0,C 180,E1 9921.086,E2 9921.086} C_VEL
LIN {X 0,Y 178.718,Z 1189.782,A -85,B 0,C 180,E1 9913.207,E2 9913.207} C_VEL
LIN {X 0,Y 176.873,Z 1184.539,A -85,B 0,C 180,E1 9906.173,E2 9906.173} C_VEL
LIN {X 0,Y 176.432,Z 1178.723,A -85,B 0,C 180,E1 9900.007,E2 9900.007} C_VEL
LIN {X 0,Y 176.491,Z 1171.729,A -85,B 0,C 180,E1 9894.154,E2 9894.154} C_VEL
LIN {X 0,Y 177.084,Z 1163.71,A -85,B 0,C 180,E1 9888.609,E2 9888.609} C_VEL
LIN {X 0,Y 178.771,Z 1152.868,A -85,B 0,C 180,E1 9882.428,E2 9882.428} C_VEL
LIN {X 0,Y 181.606,Z 1140.658,A -85,B 0,C 180,E1 9876.653,E2 9876.653} C_VEL
LIN {X 0,Y 185.771,Z 1126.194,A -85,B 0,C 180,E1 9871.034,E2 9871.034} C_VEL
LIN {X 0,Y 191.169,Z 1109.435,A -85,B 0,C 180,E1 9865.737,E2 9865.737} C_VEL
LIN {X 0,Y 197.096,Z 1091.808,A -85,B 0,C 180,E1 9861.215,E2 9861.215} C_VEL
LIN {X 0,Y 203.384,Z 1073.074,A -85,B 0,C 180,E1 9857.287,E2 9857.287} C_VEL
LIN {X 0,Y 210.196,Z 1052.013,A -85,B 0,C 180,E1 9853.703,E2 9853.703} C_VEL
LIN {X 0,Y 216.882,Z 1029.687,A -85,B 0,C 180,E1 9850.657,E2 9850.657} C_VEL
LIN {X 0,Y 223.135,Z 1006.654,A -85,B 0,C 180,E1 9848.158,E2 9848.158} C_VEL
LIN {X 0,Y 228.869,Z 982.465,A -85,B 0,C 180,E1 9846.087,E2 9846.087} C_VEL
LIN {X 0,Y 233.842,Z 957.624,A -85,B 0,C 180,E1 9844.449,E2 9844.449} C_VEL
LIN {X 0,Y 238.205,Z 930.386,A -85,B 0,C 180,E1 9843.115,E2 9843.115} C_VEL
LIN {X 0,Y 257.274,Z 803.913,A -85,B 0,C 180,E1 9838.054,E2 9838.054} C_VEL
LIN {X 0,Y 244.596,Z 779.407,A -85,B 0,C 180,E1 9833.78,E2 9833.78} C_VEL
LIN {X 0,Y 233.223,Z 758.527,A -85,B 0,C 180,E1 9829.45,E2 9829.45} C_VEL
LIN {X 0,Y 222.635,Z 740.499,A -85,B 0,C 180,E1 9824.969,E2 9824.969} C_VEL
LIN {X 0,Y 213.208,Z 725.182,A -85,B 0,C 180,E1 9820.406,E2 9820.406} C_VEL
LIN {X 0,Y 204.568,Z 711.97,A -85,B 0,C 180,E1 9815.684,E2 9815.684} C_VEL
LIN {X 0,Y 199.619,Z 705.17,A -85,B 0,C 180,E1 9812.731,E2 9812.731} C_VEL
LIN {X 0,Y 196.983,Z 701.297,A -85,B 0,C 180,E1 9811.011,E2 9811.011} C_VEL
LIN {X 0,Y 193.938,Z 696.899,A -85,B 0,C 180,E1 9808.863,E2 9808.863} C_VEL
LIN {X 0,Y 190.128,Z 691.979,A -85,B 0,C 180,E1 9806.084,E2 9806.084} C_VEL
LIN {X 0,Y 189.199,Z 690.342,A -85,B 0,C 180,E1 9805.306,E2 9805.306} C_VEL
LIN {X 0,Y 186.254,Z 687.208,A -85,B 0,C 180,E1 9802.997,E2 9802.997} C_VEL
LIN {X 0,Y 184.911,Z 684.448,A -85,B 0,C 180,E1 9801.609,E2 9801.609} C_VEL
LIN {X 0,Y 181.848,Z 681.931,A -85,B 0,C 180,E1 9798.989,E2 9798.989} C_VEL
LIN {X 0,Y 180.421,Z 678.789,A -85,B 0,C 180,E1 9797.302,E2 9797.302} C_VEL
LIN {X 0,Y 180.324,Z 678.173,A -85,B 0,C 180,E1 9797.027,E2 9797.027} C_VEL
LIN {X 0,Y 180.315,Z 678.247,A -85,B 0,C 180,E1 9795.801,E2 9795.801} C_VEL
LIN {X 0,Y 181.29,Z 681.15,A -85,B 0,C 180,E1 9794.981,E2 9794.981} C_VEL
LIN {X 0,Y 186.733,Z 693.202,A -85,B 0,C 180,E1 9791.426,E2 9791.426} C_VEL
LIN {X 0,Y 193.212,Z 709.842,A -85,B 0,C 180,E1 9787.078,E2 9787.078} C_VEL
LIN {X 0,Y 199.488,Z 728.693,A -85,B 0,C 180,E1 9782.707,E2 9782.707} C_VEL
LIN {X 0,Y 205.284,Z 748.351,A -85,B 0,C 180,E1 9778.594,E2 9778.594} C_VEL
LIN {X 0,Y 208.226,Z 759.99,A -85,B 0,C 180,E1 9776.32,E2 9776.32} C_VEL
LIN {X 0,Y 201.827,Z 803.205,A -85,B 0,C 180,E1 9770.354,E2 9770.354} C_VEL
LIN {X 0,Y 195.679,Z 849.325,A -85,B 0,C 180,E1 9763.789,E2 9763.789} C_VEL
LIN {X 0,Y 192.125,Z 870.728,A -85,B 0,C 180,E1 9760.851,E2 9760.851} C_VEL
LIN {X 0,Y 185.509,Z 984.111,A -85,B 0,C 180,E1 9753.948,E2 9753.948} C_VEL
LIN {X 0,Y 184.216,Z 1019.332,A -85,B 0,C 180,E1 9751.578,E2 9751.578} C_VEL
LIN {X 0,Y 183.157,Z 1037.298,A -85,B 0,C 180,E1 9749.779,E2 9749.779} C_VEL
LIN {X 0,Y 181.82,Z 1055.071,A -85,B 0,C 180,E1 9747.327,E2 9747.327} C_VEL
LIN {X 0,Y 180.523,Z 1071.047,A -85,B 0,C 180,E1 9744.447,E2 9744.447} C_VEL
LIN {X 0,Y 179.415,Z 1085.242,A -85,B 0,C 180,E1 9741.23,E2 9741.23} C_VEL
LIN {X 0,Y 178.577,Z 1099.302,A -85,B 0,C 180,E1 9737.255,E2 9737.255} C_VEL
LIN {X 0,Y 178.265,Z 1111.461,A -85,B 0,C 180,E1 9732.958,E2 9732.958} C_VEL
LIN {X 0,Y 178.593,Z 1121.298,A -85,B 0,C 180,E1 9728.687,E2 9728.687} C_VEL
LIN {X 0,Y 179.884,Z 1130.302,A -85,B 0,C 180,E1 9723.818,E2 9723.818} C_VEL
LIN {X 0,Y 182.312,Z 1137.374,A -85,B 0,C 180,E1 9719.05,E2 9719.05} C_VEL
LIN {X 0,Y 186.255,Z 1142.854,A -85,B 0,C 180,E1 9714.139,E2 9714.139} C_VEL
LIN {X 0,Y 191.601,Z 1146.698,A -85,B 0,C 180,E1 9709.469,E2 9709.469} C_VEL
LIN {X 0,Y 198.274,Z 1148.727,A -85,B 0,C 180,E1 9705.09,E2 9705.09} C_VEL
LIN {X 0,Y 206.704,Z 1149.017,A -85,B 0,C 180,E1 9700.79,E2 9700.79} C_VEL
LIN {X 0,Y 215.762,Z 1147.535,A -85,B 0,C 180,E1 9697.085,E2 9697.085} C_VEL
LIN {X 0,Y 226.418,Z 1143.992,A -85,B 0,C 180,E1 9693.505,E2 9693.505} C_VEL
LIN {X 0,Y 236.594,Z 1139.128,A -85,B 0,C 180,E1 9690.638,E2 9690.638} C_VEL
LIN {X 0,Y 248.13,Z 1131.909,A -85,B 0,C 180,E1 9687.86,E2 9687.86} C_VEL
LIN {X 0,Y 258.728,Z 1123.68,A -85,B 0,C 180,E1 9685.646,E2 9685.646} C_VEL
LIN {X 0,Y 245.402,Z 1134.734,A -85,B 0,C 180,E1 9683.38,E2 9683.38} C_VEL
LIN {X 0,Y 231.158,Z 1145.171,A -85,B 0,C 180,E1 9680.343,E2 9680.343} C_VEL
LIN {X 0,Y 218.136,Z 1153.715,A -85,B 0,C 180,E1 9676.782,E2 9676.782} C_VEL
LIN {X 0,Y 206.134,Z 1160.727,A -85,B 0,C 180,E1 9672.49,E2 9672.49} C_VEL
LIN {X 0,Y 195.721,Z 1166.157,A -85,B 0,C 180,E1 9667.435,E2 9667.435} C_VEL
LIN {X 0,Y 193.749,Z 1167.122,A -85,B 0,C 180,E1 9666.243,E2 9666.243} C_VEL
LIN {X 0,Y 189.44,Z 1168.586,A -85,B 0,C 180,E1 9664.152,E2 9664.152} C_VEL
LIN {X 0,Y 179.201,Z 1170.107,A -85,B 0,C 180,E1 9660.049,E2 9660.049} C_VEL
LIN {X 0,Y 175.425,Z 1170.36,A -85,B 0,C 180,E1 9657.658,E2 9657.658} C_VEL
LIN {X 0,Y 174.801,Z 1170.439,A -85,B 0,C 180,E1 9656.964,E2 9656.964} C_VEL
LIN {X 0,Y 171.541,Z 1170.196,A -85,B 0,C 180,E1 9650.19,E2 9650.19} C_VEL
LIN {X 0,Y 171.063,Z 1169.666,A -85,B 0,C 180,E1 9647.163,E2 9647.163} C_VEL
LIN {X 0,Y 169.913,Z 1180.082,A -85,B 0,C 180,E1 9640.506,E2 9640.506} C_VEL
LIN {X 0,Y 169.972,Z 1186.957,A -85,B 0,C 180,E1 9635.058,E2 9635.058} C_VEL
LIN {X 0,Y 170.077,Z 1191.749,A -85,B 0,C 180,E1 9630.332,E2 9630.332} C_VEL
LIN {X 0,Y 169.58,Z 1195.345,A -85,B 0,C 180,E1 9625.599,E2 9625.599} C_VEL
LIN {X 0,Y 169.181,Z 1199.147,A -85,B 0,C 180,E1 9618.403,E2 9618.403} C_VEL
LIN {X 0,Y 171.159,Z 1201.718,A -85,B 0,C 180,E1 9610.19,E2 9610.19} C_VEL
LIN {X 0,Y 177.9,Z 1202.867,A -85,B 0,C 180,E1 9600.722,E2 9600.722} C_VEL
LIN {X 0,Y 188.626,Z 1202.269,A -85,B 0,C 180,E1 9592.677,E2 9592.677} C_VEL
LIN {X 0,Y 204.475,Z 1199.944,A -85,B 0,C 180,E1 9585.233,E2 9585.233} C_VEL
LIN {X 0,Y 211.442,Z 1198.745,A -85,B 0,C 180,E1 9582.736,E2 9582.736} C_VEL
LIN {X 0,Y 195.201,Z 1198.366,A -85,B 0,C 180,E1 9576.098,E2 9576.098} C_VEL
LIN {X 0,Y 182.376,Z 1196.32,A -85,B 0,C 180,E1 9568.139,E2 9568.139} C_VEL
LIN {X 0,Y 174.258,Z 1192.729,A -85,B 0,C 180,E1 9559.795,E2 9559.795} C_VEL
LIN {X 0,Y 170.205,Z 1187.892,A -85,B 0,C 180,E1 9551.872,E2 9551.872} C_VEL
LIN {X 0,Y 168.727,Z 1181.945,A -85,B 0,C 180,E1 9544.426,E2 9544.426} C_VEL
LIN {X 0,Y 168.471,Z 1176.11,A -85,B 0,C 180,E1 9538.647,E2 9538.647} C_VEL
LIN {X 0,Y 168.622,Z 1169.031,A -85,B 0,C 180,E1 9532.854,E2 9532.854} C_VEL
LIN {X 0,Y 169.508,Z 1159.827,A -85,B 0,C 180,E1 9526.708,E2 9526.708} C_VEL
LIN {X 0,Y 171.494,Z 1148.903,A -85,B 0,C 180,E1 9520.597,E2 9520.597} C_VEL
LIN {X 0,Y 174.818,Z 1135.861,A -85,B 0,C 180,E1 9514.606,E2 9514.606} C_VEL
LIN {X 0,Y 179.245,Z 1121.384,A -85,B 0,C 180,E1 9509.131,E2 9509.131} C_VEL
LIN {X 0,Y 184.924,Z 1104.461,A -85,B 0,C 180,E1 9503.897,E2 9503.897} C_VEL
LIN {X 0,Y 191.379,Z 1085.854,A -85,B 0,C 180,E1 9499.235,E2 9499.235} C_VEL
LIN {X 0,Y 197.858,Z 1066.937,A -85,B 0,C 180,E1 9495.386,E2 9495.386} C_VEL
LIN {X 0,Y 204.53,Z 1046.484,A -85,B 0,C 180,E1 9492.015,E2 9492.015} C_VEL
LIN {X 0,Y 211.516,Z 1023.27,A -85,B 0,C 180,E1 9488.96,E2 9488.96} C_VEL
LIN {X 0,Y 217.763,Z 1000.064,A -85,B 0,C 180,E1 9486.542,E2 9486.542} C_VEL
LIN {X 0,Y 223.57,Z 975.161,A -85,B 0,C 180,E1 9484.521,E2 9484.521} C_VEL
LIN {X 0,Y 228.537,Z 949.166,A -85,B 0,C 180,E1 9482.927,E2 9482.927} C_VEL
LIN {X 0,Y 250.688,Z 806.631,A -85,B 0,C 180,E1 9476.984,E2 9476.984} C_VEL
LIN {X 0,Y 238,Z 781.877,A -85,B 0,C 180,E1 9472.48,E2 9472.48} C_VEL
LIN {X 0,Y 227.238,Z 762.086,A -85,B 0,C 180,E1 9468.208,E2 9468.208} C_VEL
LIN {X 0,Y 217.077,Z 744.524,A -85,B 0,C 180,E1 9463.645,E2 9463.645} C_VEL
LIN {X 0,Y 208.359,Z 730.317,A -85,B 0,C 180,E1 9459.255,E2 9459.255} C_VEL
LIN {X 0,Y 200.671,Z 718.366,A -85,B 0,C 180,E1 9454.851,E2 9454.851} C_VEL
LIN {X 0,Y 193.601,Z 708.157,A -85,B 0,C 180,E1 9450.3,E2 9450.3} C_VEL
LIN {X 0,Y 189.621,Z 702.589,A -85,B 0,C 180,E1 9447.435,E2 9447.435} C_VEL
LIN {X 0,Y 186.517,Z 698.192,A -85,B 0,C 180,E1 9445.007,E2 9445.007} C_VEL
LIN {X 0,Y 182.805,Z 693.459,A -85,B 0,C 180,E1 9441.829,E2 9441.829} C_VEL
LIN {X 0,Y 181.805,Z 691.664,A -85,B 0,C 180,E1 9440.827,E2 9440.827} C_VEL
LIN {X 0,Y 178.743,Z 688.74,A -85,B 0,C 180,E1 9438.059,E2 9438.059} C_VEL
LIN {X 0,Y 177.503,Z 686.289,A -85,B 0,C 180,E1 9436.568,E2 9436.568} C_VEL
LIN {X 0,Y 176.098,Z 686.991,A -85,B 0,C 180,E1 9435.537,E2 9435.537} C_VEL
LIN {X 0,Y 175.788,Z 687.113,A -85,B 0,C 180,E1 9435.174,E2 9435.174} C_VEL
LIN {X 0,Y 182.589,Z 703.117,A -85,B 0,C 180,E1 9430.49,E2 9430.49} C_VEL
LIN {X 0,Y 188.921,Z 720.771,A -85,B 0,C 180,E1 9425.955,E2 9425.955} C_VEL
LIN {X 0,Y 194.967,Z 740.13,A -85,B 0,C 180,E1 9421.519,E2 9421.519} C_VEL
LIN {X 0,Y 200.402,Z 760.144,A -85,B 0,C 180,E1 9417.399,E2 9417.399} C_VEL
LIN {X 0,Y 200.669,Z 762.435,A -85,B 0,C 180,E1 9416.987,E2 9416.987} C_VEL
LIN {X 0,Y 194.196,Z 804.544,A -85,B 0,C 180,E1 9411.019,E2 9411.019} C_VEL
LIN {X 0,Y 187.878,Z 850.449,A -85,B 0,C 180,E1 9404.315,E2 9404.315} C_VEL
LIN {X 0,Y 184.221,Z 871.72,A -85,B 0,C 180,E1 9401.297,E2 9401.297} C_VEL
LIN {X 0,Y 177.552,Z 983.167,A -85,B 0,C 180,E1 9394.158,E2 9394.158} C_VEL
LIN {X 0,Y 176.154,Z 1020.36,A -85,B 0,C 180,E1 9391.519,E2 9391.519} C_VEL
LIN {X 0,Y 175.049,Z 1038.585,A -85,B 0,C 180,E1 9389.601,E2 9389.601} C_VEL
LIN {X 0,Y 173.705,Z 1056.186,A -85,B 0,C 180,E1 9387.04,E2 9387.04} C_VEL
LIN {X 0,Y 172.389,Z 1072.388,A -85,B 0,C 180,E1 9383.946,E2 9383.946} C_VEL
LIN {X 0,Y 171.306,Z 1086.783,A -85,B 0,C 180,E1 9380.492,E2 9380.492} C_VEL
LIN {X 0,Y 170.572,Z 1100.15,A -85,B 0,C 180,E1 9376.509,E2 9376.509} C_VEL
LIN {X 0,Y 170.359,Z 1111.848,A -85,B 0,C 180,E1 9372.191,E2 9372.191} C_VEL
LIN {X 0,Y 170.869,Z 1122.448,A -85,B 0,C 180,E1 9367.389,E2 9367.389} C_VEL
LIN {X 0,Y 172.601,Z 1131.956,A -85,B 0,C 180,E1 9361.985,E2 9361.985} C_VEL
LIN {X 0,Y 175.741,Z 1139.258,A -85,B 0,C 180,E1 9356.731,E2 9356.731} C_VEL
LIN {X 0,Y 181.225,Z 1145.329,A -85,B 0,C 180,E1 9350.94,E2 9350.94} C_VEL
LIN {X 0,Y 188.162,Z 1148.862,A -85,B 0,C 180,E1 9345.845,E2 9345.845} C_VEL
LIN {X 0,Y 196.23,Z 1150.379,A -85,B 0,C 180,E1 9341.384,E2 9341.384} C_VEL
LIN {X 0,Y 206.003,Z 1149.976,A -85,B 0,C 180,E1 9337.145,E2 9337.145} C_VEL
LIN {X 0,Y 216.077,Z 1147.86,A -85,B 0,C 180,E1 9333.62,E2 9333.62} C_VEL
LIN {X 0,Y 227.72,Z 1143.601,A -85,B 0,C 180,E1 9330.248,E2 9330.248} C_VEL
LIN {X 0,Y 239.464,Z 1137.625,A -85,B 0,C 180,E1 9327.403,E2 9327.403} C_VEL
LIN {X 0,Y 246.67,Z 1133.123,A -85,B 0,C 180,E1 9325.829,E2 9325.829} C_VEL
LIN {X 0,Y 231.524,Z 1143.539,A -85,B 0,C 180,E1 9323.025,E2 9323.025} C_VEL
LIN {X 0,Y 217.581,Z 1151.996,A -85,B 0,C 180,E1 9319.709,E2 9319.709} C_VEL
LIN {X 0,Y 204.253,Z 1159.057,A -85,B 0,C 180,E1 9315.563,E2 9315.563} C_VEL
LIN {X 0,Y 192.342,Z 1164.578,A -85,B 0,C 180,E1 9310.521,E2 9310.521} C_VEL
LIN {X 0,Y 183.123,Z 1168.214,A -85,B 0,C 180,E1 9304.976,E2 9304.976} C_VEL
LIN {X 0,Y 176.242,Z 1170.155,A -85,B 0,C 180,E1 9298.826,E2 9298.826} C_VEL
LIN {X 0,Y 174.801,Z 1170.439,A -85,B 0,C 180,E1 9296.964,E2 9296.964} C_VEL
LIN {X 0,Y 172.734,Z 1170.374,A -85,B 0,C 180,E1 9295.376,E2 9295.376} C_VEL
LIN {X 0,Y 165.149,Z 1168.564,A -85,B 0,C 180,E1 9291.542,E2 9291.542} C_VEL
LIN {X 0,Y 163.731,Z 1167.913,A -85,B 0,C 180,E1 9289.798,E2 9289.798} C_VEL
LIN {X 0,Y 163.408,Z 1167.503,A -85,B 0,C 180,E1 9287.626,E2 9287.626} C_VEL
LIN {X 0,Y 162.077,Z 1178.183,A -85,B 0,C 180,E1 9280.661,E2 9280.661} C_VEL
LIN {X 0,Y 162.176,Z 1185.602,A -85,B 0,C 180,E1 9274.592,E2 9274.592} C_VEL
LIN {X 0,Y 162.295,Z 1189.811,A -85,B 0,C 180,E1 9270.348,E2 9270.348} C_VEL
LIN {X 0,Y 161.828,Z 1193.346,A -85,B 0,C 180,E1 9265.743,E2 9265.743} C_VEL
LIN {X 0,Y 161.349,Z 1196.94,A -85,B 0,C 180,E1 9259.281,E2 9259.281} C_VEL
LIN {X 0,Y 163.148,Z 1200.24,A -85,B 0,C 180,E1 9250.296,E2 9250.296} C_VEL
LIN {X 0,Y 169.265,Z 1201.843,A -85,B 0,C 180,E1 9241.023,E2 9241.023} C_VEL
LIN {X 0,Y 181.099,Z 1201.81,A -85,B 0,C 180,E1 9231.797,E2 9231.797} C_VEL
LIN {X 0,Y 196.351,Z 1200.235,A -85,B 0,C 180,E1 9224.522,E2 9224.522} C_VEL
LIN {X 0,Y 201.086,Z 1199.584,A -85,B 0,C 180,E1 9222.67,E2 9222.67} C_VEL
LIN {X 0,Y 185.158,Z 1198.36,A -85,B 0,C 180,E1 9215.685,E2 9215.685} C_VEL
LIN {X 0,Y 173.073,Z 1195.593,A -85,B 0,C 180,E1 9207.535,E2 9207.535} C_VEL
LIN {X 0,Y 165.572,Z 1191.392,A -85,B 0,C 180,E1 9199.04,E2 9199.04} C_VEL
LIN {X 0,Y 161.86,Z 1185.878,A -85,B 0,C 180,E1 9190.688,E2 9190.688} C_VEL
LIN {X 0,Y 160.727,Z 1179.965,A -85,B 0,C 180,E1 9183.574,E2 9183.574} C_VEL
LIN {X 0,Y 160.542,Z 1173.252,A -85,B 0,C 180,E1 9177.152,E2 9177.152} C_VEL
LIN {X 0,Y 160.852,Z 1165.482,A -85,B 0,C 180,E1 9171.068,E2 9171.068} C_VEL
LIN {X 0,Y 162.178,Z 1154.994,A -85,B 0,C 180,E1 9164.268,E2 9164.268} C_VEL
LIN {X 0,Y 164.742,Z 1143.125,A -85,B 0,C 180,E1 9157.904,E2 9157.904} C_VEL
LIN {X 0,Y 168.767,Z 1129.001,A -85,B 0,C 180,E1 9151.717,E2 9151.717} C_VEL
LIN {X 0,Y 173.924,Z 1113.333,A -85,B 0,C 180,E1 9146.116,E2 9146.116} C_VEL
LIN {X 0,Y 180.374,Z 1095.032,A -85,B 0,C 180,E1 9140.816,E2 9140.816} C_VEL
LIN {X 0,Y 187.082,Z 1076.136,A -85,B 0,C 180,E1 9136.423,E2 9136.423} C_VEL
LIN {X 0,Y 193.876,Z 1056.375,A -85,B 0,C 180,E1 9132.71,E2 9132.71} C_VEL
LIN {X 0,Y 200.764,Z 1035.056,A -85,B 0,C 180,E1 9129.48,E2 9129.48} C_VEL
LIN {X 0,Y 207.475,Z 1012.266,A -85,B 0,C 180,E1 9126.736,E2 9126.736} C_VEL
LIN {X 0,Y 213.838,Z 987.607,A -85,B 0,C 180,E1 9124.417,E2 9124.417} C_VEL
LIN {X 0,Y 219.212,Z 962.998,A -85,B 0,C 180,E1 9122.631,E2 9122.631} C_VEL
LIN {X 0,Y 223.938,Z 936.416,A -85,B 0,C 180,E1 9121.203,E2 9121.203} C_VEL
LIN {X 0,Y 244.132,Z 809.279,A -85,B 0,C 180,E1 9115.864,E2 9115.864} C_VEL
LIN {X 0,Y 232.021,Z 785.48,A -85,B 0,C 180,E1 9111.359,E2 9111.359} C_VEL
LIN {X 0,Y 221.43,Z 765.781,A -85,B 0,C 180,E1 9106.937,E2 9106.937} C_VEL
LIN {X 0,Y 211.637,Z 748.808,A -85,B 0,C 180,E1 9102.348,E2 9102.348} C_VEL
LIN {X 0,Y 202.919,Z 734.213,A -85,B 0,C 180,E1 9097.649,E2 9097.649} C_VEL
LIN {X 0,Y 195.878,Z 723.533,A -85,B 0,C 180,E1 9093.443,E2 9093.443} C_VEL
LIN {X 0,Y 190.162,Z 714.956,A -85,B 0,C 180,E1 9089.552,E2 9089.552} C_VEL
LIN {X 0,Y 186.125,Z 709.272,A -85,B 0,C 180,E1 9086.539,E2 9086.539} C_VEL
LIN {X 0,Y 182.515,Z 704.142,A -85,B 0,C 180,E1 9083.556,E2 9083.556} C_VEL
LIN {X 0,Y 179.561,Z 700.117,A -85,B 0,C 180,E1 9080.873,E2 9080.873} C_VEL
LIN {X 0,Y 178.677,Z 698.78,A -85,B 0,C 180,E1 9079.986,E2 9079.986} C_VEL
LIN {X 0,Y 175.682,Z 695.523,A -85,B 0,C 180,E1 9077.088,E2 9077.088} C_VEL
LIN {X 0,Y 175.059,Z 694.654,A -85,B 0,C 180,E1 9076.386,E2 9076.386} C_VEL
LIN {X 0,Y 172.781,Z 696.87,A -85,B 0,C 180,E1 9074.91,E2 9074.91} C_VEL
LIN {X 0,Y 171.919,Z 697.17,A -85,B 0,C 180,E1 9074.141,E2 9074.141} C_VEL
LIN {X 0,Y 178.05,Z 712.623,A -85,B 0,C 180,E1 9069.667,E2 9069.667} C_VEL
LIN {X 0,Y 183.886,Z 729.937,A -85,B 0,C 180,E1 9065.253,E2 9065.253} C_VEL
LIN {X 0,Y 189.655,Z 749.403,A -85,B 0,C 180,E1 9060.817,E2 9060.817} C_VEL
LIN {X 0,Y 193.219,Z 763.892,A -85,B 0,C 180,E1 9057.796,E2 9057.796} C_VEL
LIN {X 0,Y 186.364,Z 807.108,A -85,B 0,C 180,E1 9051.517,E2 9051.517} C_VEL
LIN {X 0,Y 180.036,Z 851.388,A -85,B 0,C 180,E1 9044.846,E2 9044.846} C_VEL
LIN {X 0,Y 176.32,Z 872.516,A -85,B 0,C 180,E1 9041.76,E2 9041.76} C_VEL
LIN {X 0,Y 169.545,Z 983.645,A -85,B 0,C 180,E1 9034.265,E2 9034.265} C_VEL
LIN {X 0,Y 168.113,Z 1020.948,A -85,B 0,C 180,E1 9031.473,E2 9031.473} C_VEL
LIN {X 0,Y 166.958,Z 1039.575,A -85,B 0,C 180,E1 9029.403,E2 9029.403} C_VEL
LIN {X 0,Y 165.586,Z 1057.375,A -85,B 0,C 180,E1 9026.671,E2 9026.671} C_VEL
LIN {X 0,Y 164.302,Z 1073.24,A -85,B 0,C 180,E1 9023.483,E2 9023.483} C_VEL
LIN {X 0,Y 163.265,Z 1087.545,A -85,B 0,C 180,E1 9019.862,E2 9019.862} C_VEL
LIN {X 0,Y 162.581,Z 1101.427,A -85,B 0,C 180,E1 9015.509,E2 9015.509} C_VEL
LIN {X 0,Y 162.505,Z 1112.98,A -85,B 0,C 180,E1 9010.988,E2 9010.988} C_VEL
LIN {X 0,Y 163.23,Z 1123.527,A -85,B 0,C 180,E1 9005.97,E2 9005.97} C_VEL
LIN {X 0,Y 165.319,Z 1132.995,A -85,B 0,C 180,E1 9000.339,E2 9000.339} C_VEL
LIN {X 0,Y 168.923,Z 1140.318,A -85,B 0,C 180,E1 8994.899,E2 8994.899} C_VEL
LIN {X 0,Y 174.454,Z 1146.004,A -85,B 0,C 180,E1 8989.425,E2 8989.425} C_VEL
LIN {X 0,Y 181.199,Z 1149.595,A -85,B 0,C 180,E1 8984.634,E2 8984.634} C_VEL
LIN {X 0,Y 189.85,Z 1151.523,A -85,B 0,C 180,E1 8979.974,E2 8979.974} C_VEL
LIN {X 0,Y 199.236,Z 1151.657,A -85,B 0,C 180,E1 8976.008,E2 8976.008} C_VEL
LIN {X 0,Y 210.331,Z 1149.892,A -85,B 0,C 180,E1 8972.227,E2 8972.227} C_VEL
LIN {X 0,Y 221.689,Z 1146.479,A -85,B 0,C 180,E1 8969.052,E2 8969.052} C_VEL
LIN {X 0,Y 233.79,Z 1141.147,A -85,B 0,C 180,E1 8966.215,E2 8966.215} C_VEL
LIN {X 0,Y 234.474,Z 1140.815,A -85,B 0,C 180,E1 8966.016,E2 8966.016} C_VEL
LIN {X 0,Y 219.198,Z 1149.57,A -85,B 0,C 180,E1 8962.959,E2 8962.959} C_VEL
LIN {X 0,Y 204.784,Z 1156.705,A -85,B 0,C 180,E1 8959.177,E2 8959.177} C_VEL
LIN {X 0,Y 191.952,Z 1162.131,A -85,B 0,C 180,E1 8954.68,E2 8954.68} C_VEL
LIN {X 0,Y 180.592,Z 1166.14,A -85,B 0,C 180,E1 8949.131,E2 8949.131} C_VEL
LIN {X 0,Y 171.772,Z 1168.419,A -85,B 0,C 180,E1 8942.77,E2 8942.77} C_VEL
LIN {X 0,Y 165.944,Z 1168.881,A -85,B 0,C 180,E1 8935.705,E2 8935.705} C_VEL
LIN {X 0,Y 163.731,Z 1167.913,A -85,B 0,C 180,E1 8929.798,E2 8929.798} C_VEL
LIN {X 0,Y 162.81,Z 1168.356,A -85,B 0,C 180,E1 8927.902,E2 8927.902} C_VEL
LIN {X 0,Y 160.361,Z 1170.793,A -85,B 0,C 180,E1 8925.398,E2 8925.398} C_VEL
LIN {X 0,Y 154.816,Z 1177.307,A -85,B 0,C 180,E1 8920.057,E2 8920.057} C_VEL
LIN {X 0,Y 154.231,Z 1179.51,A -85,B 0,C 180,E1 8918.159,E2 8918.159} C_VEL
LIN {X 0,Y 154.472,Z 1185.332,A -85,B 0,C 180,E1 8912.963,E2 8912.963} C_VEL
LIN {X 0,Y 154.438,Z 1189.332,A -85,B 0,C 180,E1 8908.511,E2 8908.511} C_VEL
LIN {X 0,Y 153.753,Z 1193.098,A -85,B 0,C 180,E1 8902.897,E2 8902.897} C_VEL
LIN {X 0,Y 153.961,Z 1196.903,A -85,B 0,C 180,E1 8894.938,E2 8894.938} C_VEL
LIN {X 0,Y 158.081,Z 1199.903,A -85,B 0,C 180,E1 8884.772,E2 8884.772} C_VEL
LIN {X 0,Y 167.043,Z 1201.186,A -85,B 0,C 180,E1 8875.339,E2 8875.339} C_VEL
LIN {X 0,Y 181.622,Z 1200.762,A -85,B 0,C 180,E1 8866.619,E2 8866.619} C_VEL
LIN {X 0,Y 190.888,Z 1199.955,A -85,B 0,C 180,E1 8862.653,E2 8862.653} C_VEL
LIN {X 0,Y 174.648,Z 1197.813,A -85,B 0,C 180,E1 8854.934,E2 8854.934} C_VEL
LIN {X 0,Y 163.118,Z 1194.156,A -85,B 0,C 180,E1 8846.198,E2 8846.198} C_VEL
LIN {X 0,Y 156.337,Z 1189.039,A -85,B 0,C 180,E1 8837.118,E2 8837.118} C_VEL
LIN {X 0,Y 153.377,Z 1182.653,A -85,B 0,C 180,E1 8828.254,E2 8828.254} C_VEL
LIN {X 0,Y 152.713,Z 1176.596,A -85,B 0,C 180,E1 8821.509,E2 8821.509} C_VEL
LIN {X 0,Y 152.66,Z 1169.626,A -85,B 0,C 180,E1 8815.124,E2 8815.124} C_VEL
LIN {X 0,Y 153.297,Z 1160.501,A -85,B 0,C 180,E1 8808.343,E2 8808.343} C_VEL
LIN {X 0,Y 155.081,Z 1149.665,A -85,B 0,C 180,E1 8801.592,E2 8801.592} C_VEL
LIN {X 0,Y 158.324,Z 1136.752,A -85,B 0,C 180,E1 8794.976,E2 8794.976} C_VEL
LIN {X 0,Y 162.823,Z 1122.367,A -85,B 0,C 180,E1 8788.956,E2 8788.956} C_VEL
LIN {X 0,Y 168.899,Z 1105.043,A -85,B 0,C 180,E1 8783.061,E2 8783.061} C_VEL
LIN {X 0,Y 175.652,Z 1086.539,A -85,B 0,C 180,E1 8778.031,E2 8778.031} C_VEL
LIN {X 0,Y 182.717,Z 1066.964,A -85,B 0,C 180,E1 8773.763,E2 8773.763} C_VEL
LIN {X 0,Y 189.756,Z 1046.573,A -85,B 0,C 180,E1 8770.189,E2 8770.189} C_VEL
LIN {X 0,Y 196.799,Z 1024.442,A -85,B 0,C 180,E1 8767.103,E2 8767.103} C_VEL
LIN {X 0,Y 203.686,Z 1000.24,A -85,B 0,C 180,E1 8764.454,E2 8764.454} C_VEL
LIN {X 0,Y 209.779,Z 975.508,A -85,B 0,C 180,E1 8762.358,E2 8762.358} C_VEL
LIN {X 0,Y 215.012,Z 949.735,A -85,B 0,C 180,E1 8760.706,E2 8760.706} C_VEL
LIN {X 0,Y 237.682,Z 812.15,A -85,B 0,C 180,E1 8754.715,E2 8754.715} C_VEL
LIN {X 0,Y 226.19,Z 789.253,A -85,B 0,C 180,E1 8750.241,E2 8750.241} C_VEL
LIN {X 0,Y 216.115,Z 770.366,A -85,B 0,C 180,E1 8745.845,E2 8745.845} C_VEL
LIN {X 0,Y 206.086,Z 752.627,A -85,B 0,C 180,E1 8740.876,E2 8740.876} C_VEL
LIN {X 0,Y 198.087,Z 739.357,A -85,B 0,C 180,E1 8736.38,E2 8736.38} C_VEL
LIN {X 0,Y 191.896,Z 729.689,A -85,B 0,C 180,E1 8732.468,E2 8732.468} C_VEL
LIN {X 0,Y 186.486,Z 721.464,A -85,B 0,C 180,E1 8728.622,E2 8728.622} C_VEL
LIN {X 0,Y 182.633,Z 715.911,A -85,B 0,C 180,E1 8725.608,E2 8725.608} C_VEL
LIN {X 0,Y 179.38,Z 711.135,A -85,B 0,C 180,E1 8722.773,E2 8722.773} C_VEL
LIN {X 0,Y 176.284,Z 706.611,A -85,B 0,C 180,E1 8719.795,E2 8719.795} C_VEL
LIN {X 0,Y 173.195,Z 703.265,A -85,B 0,C 180,E1 8716.747,E2 8716.747} C_VEL
LIN {X 0,Y 170.945,Z 705.091,A -85,B 0,C 180,E1 8715.217,E2 8715.217} C_VEL
LIN {X 0,Y 168.718,Z 707.179,A -85,B 0,C 180,E1 8713.725,E2 8713.725} C_VEL
LIN {X 0,Y 167.982,Z 707.418,A -85,B 0,C 180,E1 8713.048,E2 8713.048} C_VEL
LIN {X 0,Y 173.929,Z 723.767,A -85,B 0,C 180,E1 8708.417,E2 8708.417} C_VEL
LIN {X 0,Y 179.712,Z 742.435,A -85,B 0,C 180,E1 8703.753,E2 8703.753} C_VEL
LIN {X 0,Y 184.949,Z 761.638,A -85,B 0,C 180,E1 8699.462,E2 8699.462} C_VEL
LIN {X 0,Y 185.753,Z 765.731,A -85,B 0,C 180,E1 8698.62,E2 8698.62} C_VEL
LIN {X 0,Y 178.6,Z 809.255,A -85,B 0,C 180,E1 8692.115,E2 8692.115} C_VEL
LIN {X 0,Y 172.292,Z 851.732,A -85,B 0,C 180,E1 8685.536,E2 8685.536} C_VEL
LIN {X 0,Y 168.402,Z 873.53,A -85,B 0,C 180,E1 8682.229,E2 8682.229} C_VEL
LIN {X 0,Y 161.572,Z 983.021,A -85,B 0,C 180,E1 8674.424,E2 8674.424} C_VEL
LIN {X 0,Y 160.051,Z 1021.908,A -85,B 0,C 180,E1 8671.355,E2 8671.355} C_VEL
LIN {X 0,Y 158.876,Z 1040.431,A -85,B 0,C 180,E1 8669.183,E2 8669.183} C_VEL
LIN {X 0,Y 157.532,Z 1057.78,A -85,B 0,C 180,E1 8666.369,E2 8666.369} C_VEL
LIN {X 0,Y 156.243,Z 1073.89,A -85,B 0,C 180,E1 8662.969,E2 8662.969} C_VEL
LIN {X 0,Y 155.246,Z 1088.22,A -85,B 0,C 180,E1 8659.167,E2 8659.167} C_VEL
LIN {X 0,Y 154.656,Z 1102.018,A -85,B 0,C 180,E1 8654.596,E2 8654.596} C_VEL
LIN {X 0,Y 154.685,Z 1113.209,A -85,B 0,C 180,E1 8650.043,E2 8650.043} C_VEL
LIN {X 0,Y 155.692,Z 1124.502,A -85,B 0,C 180,E1 8644.412,E2 8644.412} C_VEL
LIN {X 0,Y 157.996,Z 1133.46,A -85,B 0,C 180,E1 8638.883,E2 8638.883} C_VEL
LIN {X 0,Y 161.988,Z 1140.938,A -85,B 0,C 180,E1 8633.257,E2 8633.257} C_VEL
LIN {X 0,Y 167.228,Z 1146.12,A -85,B 0,C 180,E1 8628.263,E2 8628.263} C_VEL
LIN {X 0,Y 173.827,Z 1149.982,A -85,B 0,C 180,E1 8623.622,E2 8623.622} C_VEL
LIN {X 0,Y 182.803,Z 1152.508,A -85,B 0,C 180,E1 8618.831,E2 8618.831} C_VEL
LIN {X 0,Y 193.16,Z 1153.113,A -85,B 0,C 180,E1 8614.548,E2 8614.548} C_VEL
LIN {X 0,Y 204.707,Z 1151.887,A -85,B 0,C 180,E1 8610.755,E2 8610.755} C_VEL
LIN {X 0,Y 216.472,Z 1148.939,A -85,B 0,C 180,E1 8607.595,E2 8607.595} C_VEL
LIN {X 0,Y 222.176,Z 1146.983,A -85,B 0,C 180,E1 8606.198,E2 8606.198} C_VEL
LIN {X 0,Y 206.157,Z 1154.478,A -85,B 0,C 180,E1 8602.688,E2 8602.688} C_VEL
LIN {X 0,Y 191.411,Z 1160.2,A -85,B 0,C 180,E1 8598.324,E2 8598.324} C_VEL
LIN {X 0,Y 178.625,Z 1164.242,A -85,B 0,C 180,E1 8593.065,E2 8593.065} C_VEL
LIN {X 0,Y 168.283,Z 1166.651,A -85,B 0,C 180,E1 8586.871,E2 8586.871} C_VEL
LIN {X 0,Y 161.02,Z 1167.305,A -85,B 0,C 180,E1 8580.192,E2 8580.192} C_VEL
LIN {X 0,Y 156.981,Z 1166.391,A -85,B 0,C 180,E1 8573.254,E2 8573.254} C_VEL
LIN {X 0,Y 155.859,Z 1165.103,A -85,B 0,C 180,E1 8568.229,E2 8568.229} C_VEL
LIN {X 0,Y 154.296,Z 1175.582,A -85,B 0,C 180,E1 8561.205,E2 8561.205} C_VEL
LIN {X 0,Y 154.231,Z 1179.51,A -85,B 0,C 180,E1 8558.159,E2 8558.159} C_VEL
LIN {X 0,Y 153.546,Z 1182.062,A -85,B 0,C 180,E1 8555.873,E2 8555.873} C_VEL
LIN {X 0,Y 151.034,Z 1184.784,A -85,B 0,C 180,E1 8552.584,E2 8552.584} C_VEL
LIN {X 0,Y 146.505,Z 1188.92,A -85,B 0,C 180,E1 8546.2,E2 8546.2} C_VEL
LIN {X 0,Y 146.317,Z 1189.472,A -85,B 0,C 180,E1 8545.339,E2 8545.339} C_VEL
LIN {X 0,Y 145.863,Z 1193.493,A -85,B 0,C 180,E1 8538.127,E2 8538.127} C_VEL
LIN {X 0,Y 148.362,Z 1197.385,A -85,B 0,C 180,E1 8527.821,E2 8527.821} C_VEL
LIN {X 0,Y 155.341,Z 1199.582,A -85,B 0,C 180,E1 8518.137,E2 8518.137} C_VEL
LIN {X 0,Y 169.042,Z 1200.323,A -85,B 0,C 180,E1 8508.194,E2 8508.194} C_VEL
LIN {X 0,Y 180.784,Z 1199.883,A -85,B 0,C 180,E1 8502.659,E2 8502.659} C_VEL
LIN {X 0,Y 164.206,Z 1196.758,A -85,B 0,C 180,E1 8494.079,E2 8494.079} C_VEL
LIN {X 0,Y 153.287,Z 1192.215,A -85,B 0,C 180,E1 8484.683,E2 8484.683} C_VEL
LIN {X 0,Y 147.47,Z 1186.429,A -85,B 0,C 180,E1 8475.342,E2 8475.342} C_VEL
LIN {X 0,Y 145.179,Z 1179.572,A -85,B 0,C 180,E1 8466.335,E2 8466.335} C_VEL
LIN {X 0,Y 144.765,Z 1173.19,A -85,B 0,C 180,E1 8459.613,E2 8459.613} C_VEL
LIN {X 0,Y 144.825,Z 1166.441,A -85,B 0,C 180,E1 8453.667,E2 8453.667} C_VEL
LIN {X 0,Y 145.706,Z 1156.782,A -85,B 0,C 180,E1 8446.516,E2 8446.516} C_VEL
LIN {X 0,Y 147.945,Z 1145.171,A -85,B 0,C 180,E1 8439.434,E2 8439.434} C_VEL
LIN {X 0,Y 151.778,Z 1131.399,A -85,B 0,C 180,E1 8432.549,E2 8432.549} C_VEL
LIN {X 0,Y 157.247,Z 1115.206,A -85,B 0,C 180,E1 8425.984,E2 8425.984} C_VEL
LIN {X 0,Y 163.673,Z 1097.768,A -85,B 0,C 180,E1 8420.337,E2 8420.337} C_VEL
LIN {X 0,Y 170.593,Z 1079.366,A -85,B 0,C 180,E1 8415.551,E2 8415.551} C_VEL
LIN {X 0,Y 177.924,Z 1059.372,A -85,B 0,C 180,E1 8411.401,E2 8411.401} C_VEL
LIN {X 0,Y 185.713,Z 1036.698,A -85,B 0,C 180,E1 8407.691,E2 8407.691} C_VEL
LIN {X 0,Y 193.186,Z 1012.743,A -85,B 0,C 180,E1 8404.632,E2 8404.632} C_VEL
LIN {X 0,Y 199.946,Z 988.025,A -85,B 0,C 180,E1 8402.193,E2 8402.193} C_VEL
LIN {X 0,Y 205.793,Z 962.601,A -85,B 0,C 180,E1 8400.282,E2 8400.282} C_VEL
LIN {X 0,Y 210.761,Z 936.046,A -85,B 0,C 180,E1 8398.811,E2 8398.811} C_VEL
LIN {X 0,Y 231.206,Z 814.893,A -85,B 0,C 180,E1 8393.523,E2 8393.523} C_VEL
LIN {X 0,Y 220.123,Z 792.534,A -85,B 0,C 180,E1 8388.956,E2 8388.956} C_VEL
LIN {X 0,Y 210.331,Z 773.962,A -85,B 0,C 180,E1 8384.456,E2 8384.456} C_VEL
LIN {X 0,Y 200.895,Z 757.159,A -85,B 0,C 180,E1 8379.53,E2 8379.53} C_VEL
LIN {X 0,Y 193.488,Z 744.631,A -85,B 0,C 180,E1 8375.118,E2 8375.118} C_VEL
LIN {X 0,Y 187.414,Z 734.954,A -85,B 0,C 180,E1 8371.074,E2 8371.074} C_VEL
LIN {X 0,Y 182.513,Z 727.518,A -85,B 0,C 180,E1 8367.414,E2 8367.414} C_VEL
LIN {X 0,Y 179.263,Z 722.645,A -85,B 0,C 180,E1 8364.724,E2 8364.724} C_VEL
LIN {X 0,Y 176.083,Z 717.942,A -85,B 0,C 180,E1 8361.843,E2 8361.843} C_VEL
LIN {X 0,Y 172.738,Z 713.107,A -85,B 0,C 180,E1 8358.485,E2 8358.485} C_VEL
LIN {X 0,Y 171.196,Z 711.603,A -85,B 0,C 180,E1 8356.938,E2 8356.938} C_VEL
LIN {X 0,Y 167.684,Z 714.67,A -85,B 0,C 180,E1 8354.618,E2 8354.618} C_VEL
LIN {X 0,Y 164.892,Z 717.656,A -85,B 0,C 180,E1 8352.72,E2 8352.72} C_VEL
LIN {X 0,Y 164.038,Z 718.275,A -85,B 0,C 180,E1 8351.802,E2 8351.802} C_VEL
LIN {X 0,Y 169.453,Z 734.611,A -85,B 0,C 180,E1 8347.269,E2 8347.269} C_VEL
LIN {X 0,Y 175.103,Z 754.136,A -85,B 0,C 180,E1 8342.455,E2 8342.455} C_VEL
LIN {X 0,Y 178.311,Z 767.326,A -85,B 0,C 180,E1 8339.509,E2 8339.509} C_VEL
LIN {X 0,Y 170.823,Z 811.366,A -85,B 0,C 180,E1 8332.742,E2 8332.742} C_VEL
LIN {X 0,Y 164.586,Z 851.63,A -85,B 0,C 180,E1 8326.286,E2 8326.286} C_VEL
LIN {X 0,Y 160.485,Z 874.335,A -85,B 0,C 180,E1 8322.717,E2 8322.717} C_VEL
LIN {X 0,Y 153.595,Z 982.375,A -85,B 0,C 180,E1 8314.575,E2 8314.575} C_VEL
LIN {X 0,Y 152.011,Z 1022.417,A -85,B 0,C 180,E1 8311.225,E2 8311.225} C_VEL
LIN {X 0,Y 150.818,Z 1040.969,A -85,B 0,C 180,E1 8308.935,E2 8308.935} C_VEL
LIN {X 0,Y 149.434,Z 1058.806,A -85,B 0,C 180,E1 8305.894,E2 8305.894} C_VEL
LIN {X 0,Y 148.233,Z 1074.078,A -85,B 0,C 180,E1 8302.48,E2 8302.48} C_VEL
LIN {X 0,Y 147.264,Z 1088.735,A -85,B 0,C 180,E1 8298.395,E2 8298.395} C_VEL
LIN {X 0,Y 146.782,Z 1101.998,A -85,B 0,C 180,E1 8293.784,E2 8293.784} C_VEL
LIN {X 0,Y 146.965,Z 1114.145,A -85,B 0,C 180,E1 8288.6,E2 8288.6} C_VEL
LIN {X 0,Y 148.275,Z 1125.379,A -85,B 0,C 180,E1 8282.697,E2 8282.697} C_VEL
LIN {X 0,Y 150.988,Z 1134.329,A -85,B 0,C 180,E1 8276.955,E2 8276.955} C_VEL
LIN {X 0,Y 155.54,Z 1141.878,A -85,B 0,C 180,E1 8271.117,E2 8271.117} C_VEL
LIN {X 0,Y 161.354,Z 1147.134,A -85,B 0,C 180,E1 8266.007,E2 8266.007} C_VEL
LIN {X 0,Y 168.034,Z 1150.895,A -85,B 0,C 180,E1 8261.609,E2 8261.609} C_VEL
LIN {X 0,Y 177.605,Z 1153.612,A -85,B 0,C 180,E1 8256.784,E2 8256.784} C_VEL
LIN {X 0,Y 188.561,Z 1154.527,A -85,B 0,C 180,E1 8252.52,E2 8252.52} C_VEL
LIN {X 0,Y 200.672,Z 1153.529,A -85,B 0,C 180,E1 8248.782,E2 8248.782} C_VEL
LIN {X 0,Y 209.843,Z 1151.719,A -85,B 0,C 180,E1 8246.378,E2 8246.378} C_VEL
LIN {X 0,Y 193.939,Z 1157.644,A -85,B 0,C 180,E1 8242.551,E2 8242.551} C_VEL
LIN {X 0,Y 179.522,Z 1161.9,A -85,B 0,C 180,E1 8237.79,E2 8237.79} C_VEL
LIN {X 0,Y 167.254,Z 1164.558,A -85,B 0,C 180,E1 8232.026,E2 8232.026} C_VEL
LIN {X 0,Y 157.167,Z 1165.647,A -85,B 0,C 180,E1 8224.834,E2 8224.834} C_VEL
LIN {X 0,Y 151.689,Z 1165.033,A -85,B 0,C 180,E1 8218.327,E2 8218.327} C_VEL
LIN {X 0,Y 148.736,Z 1163.371,A -85,B 0,C 180,E1 8211.28,E2 8211.28} C_VEL
LIN {X 0,Y 148.375,Z 1162.564,A -85,B 0,C 180,E1 8208.867,E2 8208.867} C_VEL
LIN {X 0,Y 146.771,Z 1169.599,A -85,B 0,C 180,E1 8204.191,E2 8204.191} C_VEL
LIN {X 0,Y 146.459,Z 1178.828,A -85,B 0,C 180,E1 8197.053,E2 8197.053} C_VEL
LIN {X 0,Y 146.771,Z 1184.588,A -85,B 0,C 180,E1 8191.556,E2 8191.556} C_VEL
LIN {X 0,Y 146.569,Z 1188.163,A -85,B 0,C 180,E1 8187.258,E2 8187.258} C_VEL
LIN {X 0,Y 146.317,Z 1189.472,A -85,B 0,C 180,E1 8185.339,E2 8185.339} C_VEL
LIN {X 0,Y 145.176,Z 1190.976,A -85,B 0,C 180,E1 8182.609,E2 8182.609} C_VEL
LIN {X 0,Y 141.496,Z 1192.466,A -85,B 0,C 180,E1 8177.946,E2 8177.946} C_VEL
LIN {X 0,Y 139.062,Z 1193.577,A -85,B 0,C 180,E1 8173.241,E2 8173.241} C_VEL
LIN {X 0,Y 139.172,Z 1194.136,A -85,B 0,C 180,E1 8171.411,E2 8171.411} C_VEL
LIN {X 0,Y 144.501,Z 1197.287,A -85,B 0,C 180,E1 8161.023,E2 8161.023} C_VEL
LIN {X 0,Y 156.925,Z 1199.17,A -85,B 0,C 180,E1 8149.937,E2 8149.937} C_VEL
LIN {X 0,Y 170.6,Z 1199.354,A -85,B 0,C 180,E1 8142.613,E2 8142.613} C_VEL
LIN {X 0,Y 155.213,Z 1195.719,A -85,B 0,C 180,E1 8134.096,E2 8134.096} C_VEL
LIN {X 0,Y 144.79,Z 1190.589,A -85,B 0,C 180,E1 8124.487,E2 8124.487} C_VEL
LIN {X 0,Y 139.036,Z 1183.967,A -85,B 0,C 180,E1 8114.162,E2 8114.162} C_VEL
LIN {X 0,Y 137.256,Z 1177.495,A -85,B 0,C 180,E1 8105.863,E2 8105.863} C_VEL
LIN {X 0,Y 136.863,Z 1170.786,A -85,B 0,C 180,E1 8098.753,E2 8098.753} C_VEL
LIN {X 0,Y 137.072,Z 1162.502,A -85,B 0,C 180,E1 8091.62,E2 8091.62} C_VEL
LIN {X 0,Y 138.253,Z 1152.672,A -85,B 0,C 180,E1 8084.488,E2 8084.488} C_VEL
LIN {X 0,Y 141.018,Z 1140.282,A -85,B 0,C 180,E1 8077.057,E2 8077.057} C_VEL
LIN {X 0,Y 145.504,Z 1125.696,A -85,B 0,C 180,E1 8069.901,E2 8069.901} C_VEL
LIN {X 0,Y 151.125,Z 1110.044,A -85,B 0,C 180,E1 8063.701,E2 8063.701} C_VEL
LIN {X 0,Y 158.135,Z 1091.75,A -85,B 0,C 180,E1 8057.926,E2 8057.926} C_VEL
LIN {X 0,Y 165.617,Z 1072.261,A -85,B 0,C 180,E1 8053.082,E2 8053.082} C_VEL
LIN {X 0,Y 173.193,Z 1051.756,A -85,B 0,C 180,E1 8049.045,E2 8049.045} C_VEL
LIN {X 0,Y 180.765,Z 1029.731,A -85,B 0,C 180,E1 8045.612,E2 8045.612} C_VEL
LIN {X 0,Y 187.929,Z 1006.649,A -85,B 0,C 180,E1 8042.805,E2 8042.805} C_VEL
LIN {X 0,Y 194.594,Z 981.976,A -85,B 0,C 180,E1 8040.478,E2 8040.478} C_VEL
LIN {X 0,Y 200.396,Z 956.422,A -85,B 0,C 180,E1 8038.65,E2 8038.65} C_VEL
LIN {X 0,Y 206.572,Z 922.358,A -85,B 0,C 180,E1 8036.871,E2 8036.871} C_VEL
LIN {X 0,Y 224.86,Z 817.715,A -85,B 0,C 180,E1 8032.287,E2 8032.287} C_VEL
LIN {X 0,Y 213.919,Z 795.498,A -85,B 0,C 180,E1 8027.559,E2 8027.559} C_VEL
LIN {X 0,Y 204.831,Z 778.055,A -85,B 0,C 180,E1 8023.124,E2 8023.124} C_VEL
LIN {X 0,Y 195.504,Z 761.139,A -85,B 0,C 180,E1 8017.978,E2 8017.978} C_VEL
LIN {X 0,Y 187.881,Z 748.116,A -85,B 0,C 180,E1 8013.131,E2 8013.131} C_VEL
LIN {X 0,Y 181.004,Z 737.148,A -85,B 0,C 180,E1 8008.105,E2 8008.105} C_VEL
LIN {X 0,Y 175.96,Z 729.455,A -85,B 0,C 180,E1 8003.875,E2 8003.875} C_VEL
LIN {X 0,Y 172.87,Z 724.791,A -85,B 0,C 180,E1 8000.936,E2 8000.936} C_VEL
LIN {X 0,Y 169.709,Z 720.154,A -85,B 0,C 180,E1 7997.604,E2 7997.604} C_VEL
LIN {X 0,Y 169.345,Z 720.094,A -85,B 0,C 180,E1 7997.293,E2 7997.293} C_VEL
LIN {X 0,Y 166.348,Z 722.742,A -85,B 0,C 180,E1 7995.373,E2 7995.373} C_VEL
LIN {X 0,Y 163.52,Z 725.308,A -85,B 0,C 180,E1 7993.41,E2 7993.41} C_VEL
LIN {X 0,Y 160.893,Z 728.464,A -85,B 0,C 180,E1 7991.633,E2 7991.633} C_VEL
LIN {X 0,Y 159.839,Z 729.206,A -85,B 0,C 180,E1 7990.548,E2 7990.548} C_VEL
LIN {X 0,Y 165.227,Z 747.023,A -85,B 0,C 180,E1 7985.706,E2 7985.706} C_VEL
LIN {X 0,Y 170.181,Z 765.636,A -85,B 0,C 180,E1 7981.204,E2 7981.204} C_VEL
LIN {X 0,Y 170.893,Z 768.931,A -85,B 0,C 180,E1 7980.462,E2 7980.462} C_VEL
LIN {X 0,Y 163.058,Z 813.34,A -85,B 0,C 180,E1 7973.432,E2 7973.432} C_VEL
LIN {X 0,Y 156.907,Z 851.58,A -85,B 0,C 180,E1 7967.112,E2 7967.112} C_VEL
